Universal Robots URScript: samho_main_Fillet_2024_02_13.script

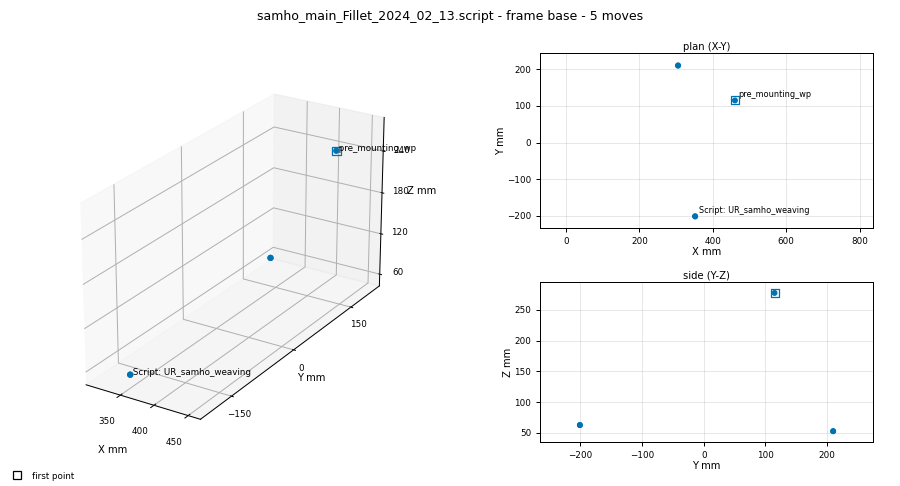
[picture p0: tool path of samho_main_Fillet_2024_02_13.script in frame base, 5 of 124 moves have a stored position in this frame; points joined in program order, loops and branches not executed]
def samho_main_Fillet_2024_02_13():
  step_count_5ae82350_5487_4ba1_a1cc_34982a72aa39 = 0.0
  thread Step_Counter_Thread_2c366939_5a87_4f2f_9225_c5964de88690():
    while (True):
      step_count_5ae82350_5487_4ba1_a1cc_34982a72aa39 = step_count_5ae82350_5487_4ba1_a1cc_34982a72aa39 + 1.0
      sync()
    end
  end
  run Step_Counter_Thread_2c366939_5a87_4f2f_9225_c5964de88690()
  modbus_add_signal("127.0.0.1", 255, 171, 2, "MODBUS_1", False)
  modbus_set_signal_update_frequency("MODBUS_1", 1)
  modbus_add_signal("127.0.0.1", 255, 153, 2, "MODBUS_2", False)
  modbus_set_signal_update_frequency("MODBUS_2", 10)
  modbus_add_signal("127.0.0.1", 255, 154, 2, "MODBUS_3", False)
  modbus_set_signal_update_frequency("MODBUS_3", 10)
  modbus_add_signal("127.0.0.1", 255, 240, 2, "MODBUS_4", False)
  modbus_set_signal_update_frequency("MODBUS_4", 10)
  set_safety_mode_transition_hardness(1)
  set_gravity([0.0, 0.0, 9.82])
  set_tool_voltage(24)
  set_tcp(p[-0.20862,-0.00524,0.38449,1.2551,0.019,-2.8747])
  set_payload(2.4, [-0.085, 0.00191, 0.125])
  set_standard_analog_input_domain(0, 1)
  set_standard_analog_input_domain(1, 1)
  set_tool_analog_input_domain(0, 1)
  set_tool_analog_input_domain(1, 1)
  set_analog_outputdomain(0, 1)
  set_analog_outputdomain(1, 1)
  set_input_actions_to_default()
  set_tool_digital_input_action(1, "freedrive")
  set_runstate_standard_digital_outputs([0])
  set_runstate_standard_digital_output_to_value(0, 1)
  set_runstate_standard_digital_output_to_value(7, 3)
  global A_Touch_trig_l=[False, True, False, True, True, True, False, True, False, False, False]
  global Auto_cur_cell=3
  global last_wv_line=p[0.52015, 0.38218, -0.0375, -1.74526, -0.73525, -1.7528]
  global Auto_trig=True
  global A_Touch_p=[p[0, 0, 0, 0, 0, 0], p[0.52015, 0.38218, -0.0375, -1.74526, -0.73525, -1.7528], p[0, 0, 0, 0, 0, 0], p[0.50413, -0.42159, 0.00426, 1.77234, -0.72849, 1.76591], p[0.52, -0.2132, 0.01111, 1.77234, -0.72849, 1.76591], p[0.51743, 0.37705, -0.04254, -1.78159, 1.77436, -0.70262], p[0, 0, 0, 0, 0, 0], p[0.52006, -0.30606, -0.04378, -1.76775, 1.766, -0.72811], p[0, 0, 0, 0, 0, 0], p[0, 0, 0, 0, 0, 0], p[0, 0, 0, 0, 0, 0], p[0, 0, 0, 0, 0, 0], p[0, 0, 0, 0, 0, 0], p[0, 0, 0, 0, 0, 0], p[0, 0, 0, 0, 0, 0], p[0, 0, 0, 0, 0, 0]]
  global last_wv_wp1=p[0.52015, 0.38218, -0.0375, -1.74526, -0.73525, -1.7528]
  global last_pose=p[0.52041, 0.38156, 0.01096, -2.11461, -0.89189, -1.42384]
  global A_Distance_list=[0, 0, 0, 0, 0, 0, 0, 0, 0, 0, 0, 0, 0, 0, 0, 0]
  global Auto_total_cell=5
  global A_Prepos_l=[p[0, 0, 0, 0, 0, 0], p[0.4924, 0.36901, -0.00027, -2.2158, -0.90076, -1.37843], p[0, 0, 0, 0, 0, 0], p[0.4524, -0.39099, 0.02973, 1.87806, -1.1242, 1.55521], p[0.4524, -0.16099, 0.02973, 1.87806, -1.1242, 1.55521], p[0.49166, 0.359, 0.00223, -2.36087, -1.03274, -1.30238], p[0, 0, 0, 0, 0, 0], p[0.45295, -0.28098, -0.02711, 2.2659, -1.09056, 1.27338], p[0, 0, 0, 0, 0, 0], p[0, 0, 0, 0, 0, 0], p[0, 0, 0, 0, 0, 0], p[0, 0, 0, 0, 0, 0], p[0, 0, 0, 0, 0, 0], p[0, 0, 0, 0, 0, 0], p[0, 0, 0, 0, 0, 0], p[0, 0, 0, 0, 0, 0]]
  global Reset_Trig=False
  global Auto_W_num=[4, 31, 32, 1, 3, 0, 0, 0, 0, 0, 0, 0, 0, 0, 0]
  global A_Speed_list=[0, 0, 0, 0, 0, 0, 0, 0, 0, 0, 0, 0, 0, 0, 0, 0]
  global last_z_bottom=-0.0502
  global last_tilt_deg=[0, -27, 0]
  global Base=p[0.0,0.0,0.0,0.0,0.0,0.0]
  global save_timer=0
  global timer_1=0
  def calculate_point_to_move_towards(feature, direction, position_distance):
    local posDir=[direction[0], direction[1], direction[2]]
    if (norm(posDir) < 1e-6):
      return get_target_waypoint()
    end
    local direction_vector_normalized=normalize(posDir)
    local displacement_pose=p[direction_vector_normalized[0] * position_distance,direction_vector_normalized[1] * position_distance,direction_vector_normalized[2] * position_distance,0,0,0]
    local wanted_displacement_in_base_frame=pose_sub(pose_trans(feature, displacement_pose), feature)
    return pose_add(get_target_waypoint(), wanted_displacement_in_base_frame)
  end
  global save_timer_is_counting=False
  global timer_1_is_counting=False
  thread Timer_Thread():
    while (True):
      if (save_timer_is_counting):
        save_timer = save_timer + get_steptime()
      end
      if (timer_1_is_counting):
        timer_1 = timer_1 + get_steptime()
      end
      sync()
    end
  end
  run Timer_Thread()
  def cell_info():
    $ 1514 "cell_info" "noBreak"
    $ 1515 "'cell_setting'"
    # 'cell_setting'
    $ 1516 "a7_f_distance≔get_center"
    global a7_f_distance=get_center
    $ 1517 "'dis + 125'"
    # 'dis + 125'
    $ 1518 "If simulation_mode"
    if (simulation_mode):
      $ 1519 "a6_f_height_l≔190"
      global a6_f_height_l=190
      $ 1520 "a6_f_height_r≔190"
      global a6_f_height_r=190
      $ 1521 "a6_f_width≔690"
      global a6_f_width=690
      $ 1522 "a6_callar_hor≔100"
      global a6_callar_hor=100
      $ 1523 "a6_callar_vert≔100"
      global a6_callar_vert=100
      $ 1524 "center_height≔50"
      global center_height=50
      $ 1525 "EXT_flag1≔integer_to_binary_list(2048)"
      global EXT_flag1= integer_to_binary_list (2048)
      $ 1526 "get_margin_z≔50"
      global get_margin_z=50
    else:
      $ 1527 "Else" "noBreak"
      $ 1528 "a6_f_height_l≔read_port_register(173)"
      global a6_f_height_l= read_port_register (173)
      $ 1529 "a6_f_height_r≔read_port_register(174)"
      global a6_f_height_r= read_port_register (174)
      $ 1530 "a6_f_width≔read_port_register(175)"
      global a6_f_width= read_port_register (175)
      $ 1531 "a6_callar_hor≔read_port_register(181)"
      global a6_callar_hor= read_port_register (181)
      $ 1532 "a6_callar_vert≔read_port_register(182)"
      global a6_callar_vert= read_port_register (182)
      $ 1533 "center_height≔read_port_register(237)"
      global center_height=read_port_register(237)
      $ 1534 "EXT_flag1≔integer_to_binary_list(read_port_register(179))"
      global EXT_flag1= integer_to_binary_list ( read_port_register (179))
      $ 1536 "get_margin_z≔read_port_register(238)"
      global get_margin_z=read_port_register(238)
      $ 1538 "If center_height>32765"
      if (center_height>32765):
        $ 1539 "center_height≔center_height-65535"
        global center_height=center_height-65535
      end
      $ 1540 "If get_margin_z>32765"
      if (get_margin_z>32765):
        $ 1541 "get_margin_z≔get_margin_z-65535"
        global get_margin_z=get_margin_z-65535
      end
    end
    $ 1542 "Initialization"
    $ 1543 "CELL_ROBOT_DIST≔a7_f_distance"
    global CELL_ROBOT_DIST=a7_f_distance
    $ 1544 "CELL_WIDTH≔a6_f_width"
    global CELL_WIDTH=a6_f_width
  end
  def robotand_cell_initalizat():
    $ 1545 "robotand_cell_initalizat" "noBreak"
    $ 1546 "If Auto_trig≟ True "
    if (Auto_trig ==   True  ):
      $ 1547 "Auto_trig≔ False "
      global Auto_trig=  False
      $ 1548 "init"
      $ 1549 "write_port_register(cell_3f_2f_151,0)"
      write_port_register(cell_3f_2f_151,0)
      $ 1550 "write_port_register(cell_info_152,0)"
      write_port_register(cell_info_152,0)
      $ 1551 "write_port_register(weld_req_153,0)"
      write_port_register(weld_req_153,0)
      $ 1552 "write_port_register(touch_cell_155,0)"
      write_port_register(touch_cell_155,0)
      $ 1553 "write_port_register(touch_num_156,0)"
      write_port_register(touch_num_156,0)
      $ 1554 "write_port_register(touch_done_157,0)"
      write_port_register(touch_done_157,0)
      $ 1555 "write_port_register(weld_done_137,0)"
      write_port_register(weld_done_137,0)
      $ 1556 "write_port_register(135,0)"
      write_port_register(135,0)
      $ 1557 "write_port_register(136,0)"
      write_port_register(136,0)
      $ 1558 "write_port_register(165,0)"
      write_port_register(165,0)
      $ 1559 "write_port_register(166,0)"
      write_port_register(166,0)
      $ 1560 "write_port_register(167,0)"
      write_port_register(167,0)
      $ 1561 "write_port_register(169,0)"
      write_port_register(169,0)
      $ 1562 "write_port_register(170,0)"
      write_port_register(170,0)
      $ 1563 "write_port_register(221,0)"
      write_port_register(221,0)
      $ 1564 "write_port_register(222,0)"
      write_port_register(222,0)
      $ 1565 "write_port_register(223,0)"
      write_port_register(223,0)
      $ 1566 "write_port_register(224,0)"
      write_port_register(224,0)
      $ 1567 "write_port_register(225,0)"
      write_port_register(225,0)
      $ 1568 "write_port_register(226,0)"
      write_port_register(226,0)
      $ 1569 "write_port_register(227,0)"
      write_port_register(227,0)
      $ 1570 "write_port_register(228,0)"
      write_port_register(228,0)
      $ 1571 "write_port_register(240,0)"
      write_port_register(240,0)
      $ 1572 "write_port_register(176,0)"
      write_port_register(176,0)
      $ 1573 "write_port_register(177,0)"
      write_port_register(177,0)
      $ 1574 "write_port_register(154,0)"
      write_port_register(154,0)
    end
    $ 1575 "sync()"
    sync()
  end
  def welding_parameter_init():
    $ 1576 "welding_parameter_init" "noBreak"
    $ 1577 "init"
    $ 1578 "If A_sel_v≟A_VL1 or A_sel_v≟A_VL2 or A_sel_v≟A_VR1 or A_sel_v≟A_VR2"
    if (A_sel_v == A_VL1  or  A_sel_v == A_VL2  or  A_sel_v == A_VR1  or  A_sel_v == A_VR2):
      $ 1579 "position_3f2f≔position_3F"
      global position_3f2f=position_3F
      $ 1580 "write_port_register(cell_3f_2f_151,A_sel_v)"
      write_port_register(cell_3f_2f_151,A_sel_v)
      $ 1581 "b8_wv_2f≔ False "
      global b8_wv_2f=  False
      $ 1582 "d_lean_degree≔0"
      global d_lean_degree=0
    else:
      $ 1583 "Else" "noBreak"
      $ 1584 "position_3f2f≔position_2F"
      global position_3f2f=position_2F
      $ 1585 "b8_wv_2f≔ True "
      global b8_wv_2f=  True
      $ 1586 "d_lean_degree≔30"
      global d_lean_degree=30
      $ 1587 "write_port_register(cell_3f_2f_151,A_HOR)"
      write_port_register(cell_3f_2f_151,A_HOR)
    end
    $ 1588 "If current_path≥2"
    if (current_path >= 2):
      $ 1589 "write_port_register(cell_info_152,current_path)"
      write_port_register(cell_info_152,current_path)
    else:
      $ 1590 "Else" "noBreak"
      $ 1591 "write_port_register(cell_info_152,1)"
      write_port_register(cell_info_152,1)
    end
    $ 1592 "write_port_register(return_done_240,0)"
    write_port_register(return_done_240,0)
    $ 1593 "Wait: 0.3"
    sleep(0.3)
    $ 1594 "write_port_register(weld_req_153,1)"
    write_port_register(weld_req_153,1)
    $ 1595 "Wait read_port_register(return_done_240)≟1"
    while (not( read_port_register (return_done_240) == 1)):
      sync()
    end
    $ 1596 "write_port_register(weld_req_153,0)"
    write_port_register(weld_req_153,0)
    $ 1597 "touch_m_check≔0"
    global touch_m_check=0
    $ 1598 "start_end_from_pendant"
    $ 1599 "d_start_current≔read_port_register(244)/10"
    global d_start_current= read_port_register (244)/10
    $ 1600 "d_start_voltage≔read_port_register(245)/10"
    global d_start_voltage= read_port_register (245)/10
    $ 1601 "d_start_time≔read_port_register(241)/10"
    global d_start_time= read_port_register (241)/10
    $ 1602 "d_end_current≔read_port_register(249)/10"
    global d_end_current= read_port_register (249)/10
    $ 1603 "d_end_voltage≔read_port_register(250)/10"
    global d_end_voltage= read_port_register (250)/10
    $ 1604 "d_end_time≔read_port_register(246)/10"
    global d_end_time= read_port_register (246)/10
    $ 1605 "d_end_current_2≔read_port_register(254)/10"
    global d_end_current_2= read_port_register (254)/10
    $ 1606 "d_end_voltage_2≔read_port_register(255)/10"
    global d_end_voltage_2= read_port_register (255)/10
    $ 1607 "d_end_time_2≔read_port_register(251)/10"
    global d_end_time_2= read_port_register (251)/10
    $ 1608 "a7_weld_crater≔[d_start_current,d_start_voltage,d_start_time,d_end_current,d_end_voltage,d_end_time,d_lean_degree]"
    global a7_weld_crater=[d_start_current,d_start_voltage,d_start_time,d_end_current,d_end_voltage,d_end_time,d_lean_degree]
    $ 1609 "a0_volt_ref≔read_port_register(231)/10"
    global a0_volt_ref= read_port_register (231)/10
    $ 1610 "a1_amp_ref≔read_port_register(232)/10"
    global a1_amp_ref= read_port_register (232)/10
    $ 1611 "a2_speed_cpm≔read_port_register(233)/10"
    global a2_speed_cpm= read_port_register (233)/10
    $ 1612 "a3_wv_amplitude≔read_port_register(234)/10"
    global a3_wv_amplitude= read_port_register (234)/10
    $ 1613 "a4_wv_frequency≔read_port_register(225)/10"
    global a4_wv_frequency= read_port_register (225)/10
    $ 1614 "b1_appro_param≔0"
    global b1_appro_param=0
    $ 1615 "b4_wv_delay2≔read_port_register(226)/10"
    global b4_wv_delay2= read_port_register (226)/10
    $ 1616 "b6_wv_delay4≔read_port_register(227)/10"
    global b6_wv_delay4= read_port_register (227)/10
    $ 1619 "b3_wv_delay1≔0"
    global b3_wv_delay1=0
    $ 1620 "b5_wv_delay3≔0"
    global b5_wv_delay3=0
    $ 1621 "b3_dealy_all≔[b3_wv_delay1,b4_wv_delay2,b5_wv_delay3,b6_wv_delay4]"
    global b3_dealy_all=[b3_wv_delay1,b4_wv_delay2,b5_wv_delay3,b6_wv_delay4]
    $ 1622 "get_width_182≔read_port_register(182)"
    global get_width_182= read_port_register (182)
    $ 1623 "b9_touch_sens≔20"
    global b9_touch_sens=20
    $ 1624 "task_angle≔register_read(228)/10"
    global task_angle=register_read(228)/10
    $ 1625 "Circle_Speed≔a2_speed_cpm"
    global Circle_Speed=a2_speed_cpm
    $ 1626 "CELL_BOTTOM≔a7_cell_bottom"
    global CELL_BOTTOM=a7_cell_bottom
    $ 1627 "a6_scallup_left≔read_port_register(176)"
    global a6_scallup_left= read_port_register (176)
    $ 1628 "a6_scallup_righ≔read_port_register(177)"
    global a6_scallup_righ= read_port_register (177)
    $ 1629 "a5_f_hole≔[a7_cell_bottom,a6_scallup_left,a6_scallup_righ]"
    global a5_f_hole=[a7_cell_bottom,a6_scallup_left,a6_scallup_righ]
    $ 1663 "폴더"
    $ 1664 "offset_2f_x≔7"
    global offset_2f_x=7
    $ 1665 "offset_3f_z≔-5"
    global offset_3f_z=-5
    $ 1666 "If A_sel_v≟A_VR1 or A_sel_v≟A_VR2"
    if (A_sel_v == A_VR1  or  A_sel_v == A_VR2):
      $ 1667 "'3F'"
      # '3F'
      $ 1668 "b2_left_par≔ False "
      global b2_left_par=  False
      $ 1669 "b8_wv_type≔1"
      global b8_wv_type=1
      $ 1670 "If A_sel_v≟A_VR2 and (b1_cell_info_R≟c or b1_cell_info_R≟d)"
      if (A_sel_v == A_VR2  and  (b1_cell_info_R == c  or  b1_cell_info_R == d)):
        $ 1671 "b7_tilt_degree≔[0,0,0]"
        global b7_tilt_degree=[0,0,0]
      else:
        $ 1672 "Else" "noBreak"
        $ 1673 "b7_tilt_degree≔[task_angle,-27,0]"
        global b7_tilt_degree=[task_angle,-27,0]
      end
      $ 1674 "c3_arc_enable≔1"
      global c3_arc_enable=1
    else:
      $ 1675 "ElseIf A_sel_v≟A_VL1 or A_sel_v≟A_VL2"
      if (A_sel_v == A_VL1  or  A_sel_v == A_VL2):
        $ 1676 "'3F'"
        # '3F'
        $ 1677 "b2_left_par≔ True "
        global b2_left_par=  True
        $ 1678 "b8_wv_type≔1"
        global b8_wv_type=1
        $ 1679 "If A_sel_v≟A_VL2 and (b1_cell_info_L≟c or b1_cell_info_L≟d)"
        if (A_sel_v == A_VL2  and  (b1_cell_info_L == c  or  b1_cell_info_L == d)):
          $ 1680 "b7_tilt_degree≔[0,0,0]"
          global b7_tilt_degree=[0,0,0]
        else:
          $ 1681 "Else" "noBreak"
          $ 1682 "b7_tilt_degree≔[task_angle,-27,0]"
          global b7_tilt_degree=[task_angle,-27,0]
        end
        $ 1683 "c3_arc_enable≔1"
        global c3_arc_enable=1
      else:
        $ 1684 "Else" "noBreak"
        $ 1685 "b2_left_par≔ True "
        global b2_left_par=  True
        $ 1686 "b8_wv_type≔2"
        global b8_wv_type=2
        $ 1687 "If A_sel_v≟A_HOR"
        if (A_sel_v == A_HOR):
          $ 1688 "b7_tilt_degree≔[30,-1*task_angle,0]"
          global b7_tilt_degree=[30,-1*task_angle,0]
        else:
          $ 1689 "Else" "noBreak"
          $ 1691 "b7_tilt_degree≔[30,-1*task_angle,0]"
          global b7_tilt_degree=[30,-1*task_angle,0]
        end
        $ 1693 "c3_arc_enable≔0"
        global c3_arc_enable=0
      end
    end
    $ 1694 "If A_sel_v≟A_VL2 or A_sel_v≟A_VR2"
    if (A_sel_v == A_VL2  or  A_sel_v == A_VR2):
      $ 1695 "If b1_cell_info_L≟E or b1_cell_info_L≟e or b1_cell_info_R≟E or b1_cell_info_R≟e"
      if (b1_cell_info_L == E  or  b1_cell_info_L == e  or  b1_cell_info_R == E  or  b1_cell_info_R == e):
        $ 1696 "a8_wv_distance≔read_port_register(182)-a5_f_hole[1]-offset_3f_begin"
        global a8_wv_distance= read_port_register (182)-a5_f_hole[1]-offset_3f_begin
      else:
        $ 1697 "Else" "noBreak"
        $ 1698 "a8_wv_distance≔read_port_register(182)-offset_3f_begin"
        global a8_wv_distance= read_port_register (182)-offset_3f_begin
      end
    else:
      $ 1703 "Else" "noBreak"
      $ 1704 "If b2_left_par"
      if (b2_left_par):
        $ 1705 "Comment"
        # Comment
        $ 1706 "a8_wv_distance≔a6_f_height_l-a5_f_hole[1]-offset_3f_begin"
        global a8_wv_distance=a6_f_height_l-a5_f_hole[1]-offset_3f_begin
        $ 1707 "Comment"
        # Comment
      else:
        $ 1708 "Else" "noBreak"
        $ 1709 "a8_wv_distance≔a6_f_height_r-a5_f_hole[1]-offset_3f_begin"
        global a8_wv_distance=a6_f_height_r-a5_f_hole[1]-offset_3f_begin
      end
    end
    $ 1710 "Ext fun & Squash"
    $ 1711 "If (A_sel_v≟A_VL1 or A_sel_v≟A_VL2) and (b1_cell_info_L≟B or b1_cell_info_L≟D)"
    if ((A_sel_v == A_VL1  or  A_sel_v == A_VL2)  and  (b1_cell_info_L == B  or  b1_cell_info_L == D)):
      $ 1712 "Scallup_check≔ True "
      global Scallup_check=  True
    else:
      $ 1713 "ElseIf (A_sel_v≟A_VR1 or A_sel_v≟A_VR2) and (b1_cell_info_R≟B or b1_cell_info_R≟D)"
      if ((A_sel_v == A_VR1  or  A_sel_v == A_VR2)  and  (b1_cell_info_R == B  or  b1_cell_info_R == D)):
        $ 1714 "Scallup_check≔ True "
        global Scallup_check=  True
      else:
        $ 1715 "Else" "noBreak"
        $ 1716 "Scallup_check≔ False "
        global Scallup_check=  False
      end
    end
    $ 1717 "'squash'"
    # 'squash'
    $ 1718 "If (EXT_flag1[7]≟ True ) and (A_sel_v≠A_HOR) and (A_sel_v≠A_VL2) and (A_sel_v≠A_VR2) and (Scallup_check≟ False ) and (A_sel_v≟A_VL1 and b1_cell_info_L≠E and b1_cell_info_L≠e) and (A_sel_v≟A_VR1 and b1_cell_info_R≠E and b1_cell_info_R≠e)"
    if ((EXT_flag1[7] ==   True  )  and  (A_sel_v != A_HOR)  and  (A_sel_v != A_VL2)  and  (A_sel_v != A_VR2)  and  (Scallup_check ==   False  )  and  (A_sel_v == A_VL1  and  b1_cell_info_L != E  and  b1_cell_info_L != e)  and  (A_sel_v == A_VR1  and  b1_cell_info_R != E  and  b1_cell_info_R != e)):
      $ 1719 "squash"
      $ 1720 "squash_enable≔1"
      global squash_enable=1
      $ 1721 "squash_voltage≔24.5"
      global squash_voltage=24.5
      $ 1722 "squash_current≔190"
      global squash_current=190
      $ 1723 "squash_amp≔7"
      global squash_amp=7
      $ 1724 "squash_speed≔10"
      global squash_speed=10
      $ 1725 "squash_cycle≔8"
      global squash_cycle=8
    else:
      $ 1726 "Else" "noBreak"
      $ 1727 "squash"
      $ 1728 "squash_enable≔0"
      global squash_enable=0
      $ 1729 "squash_voltage≔0"
      global squash_voltage=0
      $ 1730 "squash_current≔0"
      global squash_current=0
      $ 1731 "squash_amp≔0"
      global squash_amp=0
      $ 1732 "squash_speed≔0"
      global squash_speed=0
      $ 1733 "squash_cycle≔0"
      global squash_cycle=0
    end
    $ 1734 "'sladge'"
    # 'sladge'
    $ 1735 "If EXT_flag1[8]≟ True  and EXT_flag1[9]≟ False "
    if (EXT_flag1[8] ==   True    and  EXT_flag1[9] ==   False  ):
      $ 1736 "sludge≔1"
      global sludge=1
    else:
      $ 1737 "ElseIf EXT_flag1[8]≟ False  and EXT_flag1[9]≟ True "
      if (EXT_flag1[8] ==   False    and  EXT_flag1[9] ==   True  ):
        $ 1738 "sludge≔2"
        global sludge=2
      else:
        $ 1739 "Else" "noBreak"
        $ 1740 "sludge≔0"
        global sludge=0
      end
    end
    $ 1741 "waste_cycle≔2"
    global waste_cycle=2
    $ 1742 "c0_offset_x≔read_port_register(229)/10"
    global c0_offset_x= read_port_register (229)/10
    $ 1743 "c0_offset_z≔read_port_register(230)/10"
    global c0_offset_z= read_port_register (230)/10
    $ 1744 "squash_l≔[a0_volt_ref,a1_amp_ref,squash_enable,squash_voltage,squash_current,squash_amp,squash_speed,squash_cycle,waste_cycle,c0_offset_x,c0_offset_z]"
    global squash_l=[a0_volt_ref,a1_amp_ref,squash_enable,squash_voltage,squash_current,squash_amp,squash_speed,squash_cycle,waste_cycle,c0_offset_x,c0_offset_z]
    $ 1745 "WV_gap"
    $ 1746 "c5_wv_gap_y≔read_port_register(236)/10"
    global c5_wv_gap_y= read_port_register (236)/10
    $ 1747 "c6_wv_gap_cpm≔read_port_register(235)/10"
    global c6_wv_gap_cpm= read_port_register (235)/10
    $ 1748 "c9_wv_gap_freq≔a4_wv_frequency"
    global c9_wv_gap_freq=a4_wv_frequency
    $ 1749 "If c6_wv_gap_cpm≟a2_speed_cpm and a3_wv_amplitude≟c5_wv_gap_y"
    if (c6_wv_gap_cpm == a2_speed_cpm  and  a3_wv_amplitude == c5_wv_gap_y):
      $ 1750 "c4_gap_enable≔0"
      global c4_gap_enable=0
    else:
      $ 1751 "Else" "noBreak"
      $ 1752 "c4_gap_enable≔1"
      global c4_gap_enable=1
    end
    $ 1753 "c7_wv_gap≔[c4_gap_enable,c5_wv_gap_y,c6_wv_gap_cpm,c9_wv_gap_freq]"
    global c7_wv_gap=[c4_gap_enable,c5_wv_gap_y,c6_wv_gap_cpm,c9_wv_gap_freq]
    $ 1754 "arc_sen"
    $ 1755 "c3_X_p_gain≔read_port_register(186)/10"
    global c3_X_p_gain= read_port_register (186)/10
    $ 1756 "c3_X_i_gain≔read_port_register(187)/10"
    global c3_X_i_gain= read_port_register (187)/10
    $ 1757 "c3_Z_p_gain≔read_port_register(184)/10"
    global c3_Z_p_gain= read_port_register (184)/10
    $ 1758 "c3_Z_i_gain≔read_port_register(185)/10"
    global c3_Z_i_gain= read_port_register (185)/10
    $ 1759 "c3_wv_arc_fix≔0"
    global c3_wv_arc_fix=0
    $ 1760 "c3_wv_arc≔[c3_arc_enable,c3_X_p_gain,c3_X_i_gain,c3_Z_p_gain,c3_Z_i_gain,c3_wv_arc_fix]"
    global c3_wv_arc=[c3_arc_enable,c3_X_p_gain,c3_X_i_gain,c3_Z_p_gain,c3_Z_i_gain,c3_wv_arc_fix]
    $ 1761 "volt and current"
    $ 1762 "set_current_voltage(a1_amp_ref,a0_volt_ref)"
    set_current_voltage(a1_amp_ref,a0_volt_ref)
    $ 1763 "write_port_register(154,1)"
    write_port_register(154,1)
    $ 1764 "Wait read_port_register(return_done_240)≟0"
    while (not( read_port_register (return_done_240) == 0)):
      sync()
    end
    $ 1765 "write_port_register(154,0)"
    write_port_register(154,0)
  end
  def welding_parameter_sim():
    $ 1766 "welding_parameter_sim" "noBreak"
    $ 1767 "init"
    $ 1768 "If A_sel_v≟A_VL1 or A_sel_v≟A_VL2 or A_sel_v≟A_VR1 or A_sel_v≟A_VR2"
    if (A_sel_v == A_VL1  or  A_sel_v == A_VL2  or  A_sel_v == A_VR1  or  A_sel_v == A_VR2):
      $ 1769 "position_3f2f≔position_3F"
      global position_3f2f=position_3F
      $ 1770 "write_port_register(cell_3f_2f_151,A_sel_v)"
      write_port_register(cell_3f_2f_151,A_sel_v)
      $ 1771 "b8_wv_2f≔ False "
      global b8_wv_2f=  False
      $ 1772 "d_lean_degree≔0"
      global d_lean_degree=0
    else:
      $ 1773 "Else" "noBreak"
      $ 1774 "position_3f2f≔position_2F"
      global position_3f2f=position_2F
      $ 1775 "b8_wv_2f≔ True "
      global b8_wv_2f=  True
      $ 1776 "d_lean_degree≔30"
      global d_lean_degree=30
      $ 1777 "write_port_register(cell_3f_2f_151,A_HOR)"
      write_port_register(cell_3f_2f_151,A_HOR)
    end
    $ 1778 "If current_path≥2"
    if (current_path >= 2):
      $ 1779 "write_port_register(cell_info_152,current_path)"
      write_port_register(cell_info_152,current_path)
    else:
      $ 1780 "Else" "noBreak"
      $ 1781 "write_port_register(cell_info_152,1)"
      write_port_register(cell_info_152,1)
    end
    $ 1782 "write_port_register(return_done_240,0)"
    write_port_register(return_done_240,0)
    $ 1783 "Wait: 0.3"
    sleep(0.3)
    $ 1784 "write_port_register(weld_req_153,1)"
    write_port_register(weld_req_153,1)
    $ 1786 "write_port_register(weld_req_153,0)"
    write_port_register(weld_req_153,0)
    $ 1787 "touch_m_check≔0"
    global touch_m_check=0
    $ 1788 "start_end_from_pendant"
    $ 1789 "d_start_current≔read_port_register(244)/10"
    global d_start_current= read_port_register (244)/10
    $ 1790 "d_start_voltage≔read_port_register(245)/10"
    global d_start_voltage= read_port_register (245)/10
    $ 1791 "d_start_time≔read_port_register(241)/10"
    global d_start_time= read_port_register (241)/10
    $ 1792 "d_end_current≔read_port_register(249)/10"
    global d_end_current= read_port_register (249)/10
    $ 1793 "d_end_voltage≔read_port_register(250)/10"
    global d_end_voltage= read_port_register (250)/10
    $ 1794 "d_end_time≔read_port_register(246)/10"
    global d_end_time= read_port_register (246)/10
    $ 1795 "d_end_current_2≔read_port_register(254)/10"
    global d_end_current_2= read_port_register (254)/10
    $ 1796 "d_end_voltage_2≔read_port_register(255)/10"
    global d_end_voltage_2= read_port_register (255)/10
    $ 1797 "d_end_time_2≔read_port_register(251)/10"
    global d_end_time_2= read_port_register (251)/10
    $ 1798 "a7_weld_crater≔[d_start_current,d_start_voltage,d_start_time,d_end_current,d_end_voltage,d_end_time,d_lean_degree]"
    global a7_weld_crater=[d_start_current,d_start_voltage,d_start_time,d_end_current,d_end_voltage,d_end_time,d_lean_degree]
    $ 1799 "a0_volt_ref≔read_port_register(231)/10"
    global a0_volt_ref= read_port_register (231)/10
    $ 1800 "a1_amp_ref≔read_port_register(232)/10"
    global a1_amp_ref= read_port_register (232)/10
    $ 1801 "b1_appro_param≔0"
    global b1_appro_param=0
    $ 1802 "Folder"
    $ 1803 "a2_speed_cpm≔17"
    global a2_speed_cpm=17
    $ 1804 "a3_wv_amplitude≔5"
    global a3_wv_amplitude=5
    $ 1805 "a4_wv_frequency≔1.4"
    global a4_wv_frequency=1.4
    $ 1806 "b4_wv_delay2≔0.3"
    global b4_wv_delay2=0.3
    $ 1807 "b6_wv_delay4≔0.3"
    global b6_wv_delay4=0.3
    $ 1808 "b9_touch_sens≔10"
    global b9_touch_sens=10
    $ 1809 "task_angle≔0"
    global task_angle=0
    $ 1810 "a6_scallup_left≔0"
    global a6_scallup_left=0
    $ 1811 "a6_scallup_righ≔0"
    global a6_scallup_righ=0
    $ 1812 "b3_wv_delay1≔0"
    global b3_wv_delay1=0
    $ 1813 "b5_wv_delay3≔0"
    global b5_wv_delay3=0
    $ 1814 "b3_dealy_all≔[b3_wv_delay1,b4_wv_delay2,b5_wv_delay3,b6_wv_delay4]"
    global b3_dealy_all=[b3_wv_delay1,b4_wv_delay2,b5_wv_delay3,b6_wv_delay4]
    $ 1815 "get_width_182≔a6_callar_vert"
    global get_width_182=a6_callar_vert
    $ 1816 "task_angle≔register_read(228)/10"
    global task_angle=register_read(228)/10
    $ 1817 "Circle_Speed≔a2_speed_cpm"
    global Circle_Speed=a2_speed_cpm
    $ 1818 "CELL_BOTTOM≔a7_cell_bottom"
    global CELL_BOTTOM=a7_cell_bottom
    $ 1819 "a5_f_hole≔[a7_cell_bottom,a6_scallup_left,a6_scallup_righ]"
    global a5_f_hole=[a7_cell_bottom,a6_scallup_left,a6_scallup_righ]
    $ 1820 "폴더"
    $ 1821 "offset_2f_x≔7"
    global offset_2f_x=7
    $ 1822 "offset_3f_z≔-5"
    global offset_3f_z=-5
    $ 1823 "If A_sel_v≟A_VR1 or A_sel_v≟A_VR2"
    if (A_sel_v == A_VR1  or  A_sel_v == A_VR2):
      $ 1824 "'3F'"
      # '3F'
      $ 1825 "b2_left_par≔ False "
      global b2_left_par=  False
      $ 1826 "b8_wv_type≔1"
      global b8_wv_type=1
      $ 1827 "b7_tilt_degree≔[task_angle,-27,0]"
      global b7_tilt_degree=[task_angle,-27,0]
      $ 1828 "c3_arc_enable≔1"
      global c3_arc_enable=1
    else:
      $ 1829 "ElseIf A_sel_v≟A_VL1 or A_sel_v≟A_VL2"
      if (A_sel_v == A_VL1  or  A_sel_v == A_VL2):
        $ 1830 "'3F'"
        # '3F'
        $ 1831 "b2_left_par≔ True "
        global b2_left_par=  True
        $ 1832 "b8_wv_type≔1"
        global b8_wv_type=1
        $ 1833 "b7_tilt_degree≔[task_angle,-27,0]"
        global b7_tilt_degree=[task_angle,-27,0]
        $ 1834 "c3_arc_enable≔1"
        global c3_arc_enable=1
      else:
        $ 1835 "Else" "noBreak"
        $ 1836 "b2_left_par≔ True "
        global b2_left_par=  True
        $ 1837 "b8_wv_type≔2"
        global b8_wv_type=2
        $ 1838 "b7_tilt_degree≔[30,-1*task_angle,0]"
        global b7_tilt_degree=[30,-1*task_angle,0]
        $ 1840 "c3_arc_enable≔0"
        global c3_arc_enable=0
      end
    end
    $ 1841 "If A_sel_v≟A_VL2 or A_sel_v≟A_VR2"
    if (A_sel_v == A_VL2  or  A_sel_v == A_VR2):
      $ 1842 "a8_wv_distance≔read_port_register(182)"
      global a8_wv_distance= read_port_register (182)
    else:
      $ 1847 "Else" "noBreak"
      $ 1848 "If b2_left_par"
      if (b2_left_par):
        $ 1849 "Comment"
        # Comment
        $ 1850 "a8_wv_distance≔a6_f_height_l-a5_f_hole[1]"
        global a8_wv_distance=a6_f_height_l-a5_f_hole[1]
        $ 1851 "Comment"
        # Comment
      else:
        $ 1852 "Else" "noBreak"
        $ 1853 "a8_wv_distance≔a6_f_height_r-a5_f_hole[1]"
        global a8_wv_distance=a6_f_height_r-a5_f_hole[1]
      end
    end
    $ 1854 "Ext fun & Squash"
    $ 1855 "If (A_sel_v≟A_VL1 or A_sel_v≟A_VL2) and (b1_cell_info_L≟B or b1_cell_info_L≟D)"
    if ((A_sel_v == A_VL1  or  A_sel_v == A_VL2)  and  (b1_cell_info_L == B  or  b1_cell_info_L == D)):
      $ 1856 "Scallup_check≔ True "
      global Scallup_check=  True
    else:
      $ 1857 "ElseIf (A_sel_v≟A_VR1 or A_sel_v≟A_VR2) and (b1_cell_info_R≟B or b1_cell_info_R≟D)"
      if ((A_sel_v == A_VR1  or  A_sel_v == A_VR2)  and  (b1_cell_info_R == B  or  b1_cell_info_R == D)):
        $ 1858 "Scallup_check≔ True "
        global Scallup_check=  True
      else:
        $ 1859 "Else" "noBreak"
        $ 1860 "Scallup_check≔ False "
        global Scallup_check=  False
      end
    end
    $ 1861 "If (EXT_flag1[7]≟ True ) and (A_sel_v≠A_HOR) and (A_sel_v≠A_VL2) and (A_sel_v≠A_VR2) and (Scallup_check≟ False )"
    if ((EXT_flag1[7] ==   True  )  and  (A_sel_v != A_HOR)  and  (A_sel_v != A_VL2)  and  (A_sel_v != A_VR2)  and  (Scallup_check ==   False  )):
      $ 1862 "squash"
      $ 1863 "squash_enable≔1"
      global squash_enable=1
      $ 1864 "squash_voltage≔24.5"
      global squash_voltage=24.5
      $ 1865 "squash_current≔190"
      global squash_current=190
      $ 1866 "squash_amp≔7"
      global squash_amp=7
      $ 1867 "squash_speed≔10"
      global squash_speed=10
      $ 1868 "squash_cycle≔8"
      global squash_cycle=8
    else:
      $ 1869 "Else" "noBreak"
      $ 1870 "squash"
      $ 1871 "squash_enable≔0"
      global squash_enable=0
      $ 1872 "squash_voltage≔0"
      global squash_voltage=0
      $ 1873 "squash_current≔0"
      global squash_current=0
      $ 1874 "squash_amp≔0"
      global squash_amp=0
      $ 1875 "squash_speed≔0"
      global squash_speed=0
      $ 1876 "squash_cycle≔0"
      global squash_cycle=0
    end
    $ 1877 "waste_cycle≔2"
    global waste_cycle=2
    $ 1878 "c0_offset_x≔read_port_register(229)/10"
    global c0_offset_x= read_port_register (229)/10
    $ 1879 "c0_offset_z≔read_port_register(230)/10"
    global c0_offset_z= read_port_register (230)/10
    $ 1880 "squash_l≔[a0_volt_ref,a1_amp_ref,squash_enable,squash_voltage,squash_current,squash_amp,squash_speed,squash_cycle,waste_cycle,c0_offset_x,c0_offset_z]"
    global squash_l=[a0_volt_ref,a1_amp_ref,squash_enable,squash_voltage,squash_current,squash_amp,squash_speed,squash_cycle,waste_cycle,c0_offset_x,c0_offset_z]
    $ 1881 "WV_gap"
    $ 1882 "c5_wv_gap_y≔a3_wv_amplitude"
    global c5_wv_gap_y=a3_wv_amplitude
    $ 1883 "c6_wv_gap_cpm≔a2_speed_cpm"
    global c6_wv_gap_cpm=a2_speed_cpm
    $ 1884 "c9_wv_gap_freq≔a4_wv_frequency"
    global c9_wv_gap_freq=a4_wv_frequency
    $ 1885 "If c6_wv_gap_cpm≟a2_speed_cpm and a3_wv_amplitude≟c5_wv_gap_y"
    if (c6_wv_gap_cpm == a2_speed_cpm  and  a3_wv_amplitude == c5_wv_gap_y):
      $ 1886 "c4_gap_enable≔0"
      global c4_gap_enable=0
    else:
      $ 1887 "Else" "noBreak"
      $ 1888 "c4_gap_enable≔1"
      global c4_gap_enable=1
    end
    $ 1889 "c4_gap_enable≔0"
    global c4_gap_enable=0
    $ 1890 "c7_wv_gap≔[c4_gap_enable,c5_wv_gap_y,c6_wv_gap_cpm,c9_wv_gap_freq]"
    global c7_wv_gap=[c4_gap_enable,c5_wv_gap_y,c6_wv_gap_cpm,c9_wv_gap_freq]
    $ 1891 "arc_sen"
    $ 1892 "c3_X_p_gain≔read_port_register(186)/10"
    global c3_X_p_gain= read_port_register (186)/10
    $ 1893 "c3_X_i_gain≔read_port_register(187)/10"
    global c3_X_i_gain= read_port_register (187)/10
    $ 1894 "c3_Z_p_gain≔read_port_register(184)/10"
    global c3_Z_p_gain= read_port_register (184)/10
    $ 1895 "c3_Z_i_gain≔read_port_register(185)/10"
    global c3_Z_i_gain= read_port_register (185)/10
    $ 1896 "c3_wv_arc_fix≔0"
    global c3_wv_arc_fix=0
    $ 1897 "c3_wv_arc≔[c3_arc_enable,c3_X_p_gain,c3_X_i_gain,c3_Z_p_gain,c3_Z_i_gain,c3_wv_arc_fix]"
    global c3_wv_arc=[c3_arc_enable,c3_X_p_gain,c3_X_i_gain,c3_Z_p_gain,c3_Z_i_gain,c3_wv_arc_fix]
    $ 1898 "volt and current"
    $ 1899 "set_current_voltage(a1_amp_ref,a0_volt_ref)"
    set_current_voltage(a1_amp_ref,a0_volt_ref)
    $ 1900 "write_port_register(154,1)"
    write_port_register(154,1)
    $ 1902 "write_port_register(154,0)"
    write_port_register(154,0)
  end
  def Move_done():
    $ 1903 "Move_done" "noBreak"
    $ 1904 "write_port_register(robot_move_163,0)"
    write_port_register(robot_move_163,0)
    $ 1905 "write_port_register(robot_pose_164,0)"
    write_port_register(robot_pose_164,0)
    $ 1906 "write_port_register(robot_ready_141,1)"
    write_port_register(robot_ready_141,1)
  end
  def MoveFun():
    $ 1907 "MoveFun" "noBreak"
    $ 1908 "b_touch_pos≔A_Prepos_l[A_sel_v]"
    global b_touch_pos=A_Prepos_l[A_sel_v]
    $ 1909 "MoveL"
    $ 1910 "b_touch_pos" "breakAfter"
    movel(pose_trans(Base, b_touch_pos), a=0.35, v=0.35)
  end
  def MoveFun_cd():
    $ 1911 "MoveFun_cd" "noBreak"
    $ 1912 "b_touch_pos≔A_Prepos_l[A_sel_v]"
    global b_touch_pos=A_Prepos_l[A_sel_v]
    $ 1913 "If A_sel_v≟A_VR2 and (b1_cell_info_R≟c or b1_cell_info_R≟d)"
    if (A_sel_v == A_VR2  and  (b1_cell_info_R == c  or  b1_cell_info_R == d)):
      $ 1914 "tilt_deg≔27"
      global tilt_deg=27
      $ 1915 "tilt_deg_ry≔19"
      global tilt_deg_ry=19
      $ 1916 "tilt_deg_rz≔0"
      global tilt_deg_rz=0
    else:
      $ 1917 "Else" "noBreak"
      $ 1918 "tilt_deg≔10"
      global tilt_deg=10
      $ 1919 "tilt_deg_ry≔5"
      global tilt_deg_ry=5
      $ 1920 "tilt_deg_rz≔0"
      global tilt_deg_rz=0
    end
    $ 1921 "If b2_left_par"
    if (b2_left_par):
      $ 1922 "b_touch_pos≔pose_add(b_touch_pos, p[0,18/1000,0,0,0,0])"
      global b_touch_pos= pose_add (b_touch_pos, p[0,18/1000,0,0,0,0])
      $ 1923 "b_touch_pos≔pose_trans(b_touch_pos, p[0,0,0,d2r(-tilt_deg),d2r(-tilt_deg_ry),d2r(tilt_deg_rz)])"
      global b_touch_pos= pose_trans (b_touch_pos, p[0,0,0,d2r(-tilt_deg),d2r(-tilt_deg_ry),d2r(tilt_deg_rz)])
    else:
      $ 1924 "Else" "noBreak"
      $ 1925 "b_touch_pos≔pose_add(b_touch_pos, p[0,-18/1000,0,0,0,0])"
      global b_touch_pos= pose_add (b_touch_pos, p[0,-18/1000,0,0,0,0])
      $ 1926 "b_touch_pos≔pose_trans(b_touch_pos, p[0,0,0,d2r(tilt_deg),d2r(-tilt_deg_ry),d2r(-tilt_deg_rz)])"
      global b_touch_pos= pose_trans (b_touch_pos, p[0,0,0,d2r(tilt_deg),d2r(-tilt_deg_ry),d2r(-tilt_deg_rz)])
    end
    $ 1927 "MoveL"
    $ 1928 "b_touch_pos" "breakAfter"
    movel(pose_trans(Base, b_touch_pos), a=0.35, v=0.35)
  end
  def MoveandTouchFun_2f():
    $ 1929 "MoveandTouchFun_2f" "noBreak"
    $ 1930 "b_touch_pos≔A_Prepos_l[A_sel_v]"
    global b_touch_pos=A_Prepos_l[A_sel_v]
    $ 1931 "tilt_deg≔3"
    global tilt_deg=3
    $ 1932 "tilt_deg_ry≔3"
    global tilt_deg_ry=3
    $ 1933 "tilt_deg_rz≔0"
    global tilt_deg_rz=0
    $ 1934 "If  False "
    if (  False  ):
      $ 1935 "Wait: 0.01"
      sleep(0.01)
    else:
      $ 1936 "ElseIf A_sel_v≟A_HOR and b1_cell_info_L≟E"
      if (A_sel_v == A_HOR  and  b1_cell_info_L == E):
        $ 1937 "tilt_deg≔6"
        global tilt_deg=6
        $ 1938 "tilt_deg_ry≔-5"
        global tilt_deg_ry=-5
        $ 1939 "tilt_deg_rz≔0"
        global tilt_deg_rz=0
        $ 1940 "b_touch_pos≔pose_trans(b_touch_pos, p[0,0/1000,0,d2r(tilt_deg),d2r(-tilt_deg_ry),d2r(tilt_deg_rz)])"
        global b_touch_pos= pose_trans (b_touch_pos, p[0,0/1000,0,d2r(tilt_deg),d2r(-tilt_deg_ry),d2r(tilt_deg_rz)])
      else:
        $ 1941 "ElseIf A_sel_v≟A_HOR_R and b1_cell_info_R≟E"
        if (A_sel_v == A_HOR_R  and  b1_cell_info_R == E):
          $ 1942 "tilt_deg≔6"
          global tilt_deg=6
          $ 1943 "tilt_deg_ry≔-5"
          global tilt_deg_ry=-5
          $ 1944 "tilt_deg_rz≔0"
          global tilt_deg_rz=0
          $ 1945 "b_touch_pos≔pose_trans(b_touch_pos, p[0,0/1000,0,d2r(tilt_deg),d2r(-tilt_deg_ry),d2r(-tilt_deg_rz)])"
          global b_touch_pos= pose_trans (b_touch_pos, p[0,0/1000,0,d2r(tilt_deg),d2r(-tilt_deg_ry),d2r(-tilt_deg_rz)])
        else:
          $ 1946 "ElseIf b2_left_par"
          if (b2_left_par):
            $ 1947 "b_touch_pos≔pose_trans(b_touch_pos, p[0,0/1000,0,d2r(tilt_deg),d2r(-tilt_deg_ry),d2r(tilt_deg_rz)])"
            global b_touch_pos= pose_trans (b_touch_pos, p[0,0/1000,0,d2r(tilt_deg),d2r(-tilt_deg_ry),d2r(tilt_deg_rz)])
          else:
            $ 1948 "Else" "noBreak"
            $ 1949 "b_touch_pos≔pose_trans(b_touch_pos, p[0,0/1000,0,d2r(tilt_deg),d2r(-tilt_deg_ry),d2r(-tilt_deg_rz)])"
            global b_touch_pos= pose_trans (b_touch_pos, p[0,0/1000,0,d2r(tilt_deg),d2r(-tilt_deg_ry),d2r(-tilt_deg_rz)])
          end
        end
      end
    end
    $ 1950 "MoveL"
    $ 1951 "b_touch_pos" "breakAfter"
    movel(pose_trans(Base, b_touch_pos), a=0.35, v=0.35)
    $ 1952 "Touch_2f"
    $ 1953 "If  False "
    if (  False  ):
      $ 1954 "Wait: 0.01"
      sleep(0.01)
    else:
      $ 1955 "ElseIf A_sel_v≟A_HOR and b1_cell_info_L≟E"
      if (A_sel_v == A_HOR  and  b1_cell_info_L == E):
        $ 1956 "tilt_deg≔3"
        global tilt_deg=3
        $ 1957 "tilt_deg_ry≔3"
        global tilt_deg_ry=3
        $ 1958 "tilt_deg_rz≔0"
        global tilt_deg_rz=0
        $ 1959 "b_touch_pos2≔pose_trans(b_touch_pos, p[0,0/1000,0,d2r(tilt_deg),d2r(-tilt_deg_ry),d2r(tilt_deg_rz)])"
        global b_touch_pos2= pose_trans (b_touch_pos, p[0,0/1000,0,d2r(tilt_deg),d2r(-tilt_deg_ry),d2r(tilt_deg_rz)])
        $ 1960 "touch_result≔touch_fun_2f(b_touch_pos,b_touch_pos2,b2_left_par,b9_touch_sens)"
        global touch_result=touch_fun_2f(b_touch_pos,b_touch_pos2,b2_left_par,b9_touch_sens)
      else:
        $ 1961 "ElseIf A_sel_v≟A_HOR_R and b1_cell_info_R≟E"
        if (A_sel_v == A_HOR_R  and  b1_cell_info_R == E):
          $ 1962 "tilt_deg≔3"
          global tilt_deg=3
          $ 1963 "tilt_deg_ry≔3"
          global tilt_deg_ry=3
          $ 1964 "tilt_deg_rz≔0"
          global tilt_deg_rz=0
          $ 1965 "b_touch_pos2≔pose_trans(b_touch_pos, p[0,0/1000,0,d2r(tilt_deg),d2r(-tilt_deg_ry),d2r(-tilt_deg_rz)])"
          global b_touch_pos2= pose_trans (b_touch_pos, p[0,0/1000,0,d2r(tilt_deg),d2r(-tilt_deg_ry),d2r(-tilt_deg_rz)])
          $ 1966 "touch_result≔touch_fun_2f(b_touch_pos,b_touch_pos2,b2_left_par,b9_touch_sens)"
          global touch_result=touch_fun_2f(b_touch_pos,b_touch_pos2,b2_left_par,b9_touch_sens)
        else:
          $ 1967 "Else" "noBreak"
          $ 1968 "touch_result≔touch_fun_2f(b_touch_pos,b_touch_pos,b2_left_par,b9_touch_sens)"
          global touch_result=touch_fun_2f(b_touch_pos,b_touch_pos,b2_left_par,b9_touch_sens)
        end
      end
    end
    $ 1970 "If b2_left_par"
    if (b2_left_par):
      $ 1971 "touch_result≔pose_trans(touch_result,p[-(Touch_dis)/1000,0,0,0,0,0])"
      global touch_result= pose_trans (touch_result,p[-(Touch_dis)/1000,0,0,0,0,0])
    else:
      $ 1972 "Else" "noBreak"
      $ 1973 "touch_result≔pose_trans(touch_result,p[(Touch_dis)/1000,0,0,0,0,0])"
      global touch_result= pose_trans (touch_result,p[(Touch_dis)/1000,0,0,0,0,0])
    end
    $ 1974 "A_Touch_p[A_sel_v]=touch_result"
    A_Touch_p[A_sel_v]=touch_result
    $ 1975 "If EXT_flag1[3]≟ True "
    if (EXT_flag1[3] ==   True  ):
      $ 1976 "MoveL"
      $ 1977 "manual_tp≔tilt_2f_fun(touch_result,basic_tilt_2f,wv_direction)"
      global manual_tp=tilt_2f_fun(touch_result,basic_tilt_2f,wv_direction)
      $ 1978 "manual_tp≔pose_trans(manual_tp, p[0,0,-10/1000,0,0,0])"
      global manual_tp= pose_trans (manual_tp, p[0,0,-10/1000,0,0,0])
      $ 1979 "manual_tp" "breakAfter"
      movel(pose_trans(Base, manual_tp), a=0.3, v=0.15)
      $ 1980 "Wait: 1.5"
      sleep(1.5)
    end
  end
  def MoveandTouchFun_3f():
    $ 1981 "MoveandTouchFun_3f" "noBreak"
    $ 1982 "b_touch_pos≔A_Prepos_l[A_sel_v]"
    global b_touch_pos=A_Prepos_l[A_sel_v]
    $ 1983 "tilt_deg_ry≔0"
    global tilt_deg_ry=0
    $ 1984 "tilt_deg_rz≔0"
    global tilt_deg_rz=0
    $ 1985 "If b2_left_par"
    if (b2_left_par):
      $ 1986 "tilt_deg≔6"
      global tilt_deg=6
      $ 1987 "b_touch_pos≔pose_trans(b_touch_pos, p[0,0/1000,0,d2r(tilt_deg),d2r(tilt_deg_ry),d2r(tilt_deg_rz)])"
      global b_touch_pos= pose_trans (b_touch_pos, p[0,0/1000,0,d2r(tilt_deg),d2r(tilt_deg_ry),d2r(tilt_deg_rz)])
    else:
      $ 1988 "Else" "noBreak"
      $ 1989 "tilt_deg≔0.5"
      global tilt_deg=0.5
      $ 1990 "b_touch_pos≔pose_trans(b_touch_pos, p[0,0/1000,0,d2r(-tilt_deg),d2r(tilt_deg_ry),d2r(tilt_deg_rz)])"
      global b_touch_pos= pose_trans (b_touch_pos, p[0,0/1000,0,d2r(-tilt_deg),d2r(tilt_deg_ry),d2r(tilt_deg_rz)])
    end
    $ 2001 "move_pre"
    $ 2002 "If (b2_left_par≟ True  and point_dist(A_Prepos_l[A_HOR], A_Prepos_l[A_VL1])>0.032) or (b2_left_par≟ False  and point_dist(A_Prepos_l[A_HOR_R],A_Prepos_l[A_VR1])>0.032)"
    if ((b2_left_par ==   True    and  point_dist(A_Prepos_l[A_HOR], A_Prepos_l[A_VL1])>0.032)  or  (b2_left_par ==   False    and  point_dist(A_Prepos_l[A_HOR_R],A_Prepos_l[A_VR1])>0.032)):
      $ 2003 "if move from home"
      $ 2004 "j_cp≔get_actual_joint_positions()"
      global j_cp= get_actual_joint_positions ()
      $ 2005 "If b2_left_par"
      if (b2_left_par):
        $ 2006 "If norm(b_touch_pos[1]*1000)>300"
        if (norm(b_touch_pos[1]*1000)>300):
          $ 2007 "inner_p≔p[-15/1000,-35/1000,0,0,0,0]"
          global inner_p=p[-15/1000,-35/1000,0,0,0,0]
        else:
          $ 2008 "Else" "noBreak"
          $ 2009 "inner_p≔p[0,0,0,0,0,0]"
          global inner_p=p[0,0,0,0,0,0]
        end
        $ 2010 "j_tp≔get_inverse_kin(pose_add(b_touch_pos,inner_p),qnear=left_j)"
        global j_tp= get_inverse_kin (pose_add(b_touch_pos,inner_p),qnear=left_j)
      else:
        $ 2011 "Else" "noBreak"
        $ 2012 "If norm(b_touch_pos[1]*1000)>300"
        if (norm(b_touch_pos[1]*1000)>300):
          $ 2013 "inner_p≔p[-15/1000,35/1000,0,0,0,0]"
          global inner_p=p[-15/1000,35/1000,0,0,0,0]
        else:
          $ 2014 "Else" "noBreak"
          $ 2015 "inner_p≔p[0,0,0,0,0,0]"
          global inner_p=p[0,0,0,0,0,0]
        end
        $ 2016 "j_tp≔get_inverse_kin(pose_add(b_touch_pos,inner_p),qnear=right_j)"
        global j_tp= get_inverse_kin ( pose_add (b_touch_pos,inner_p),qnear=right_j)
      end
      $ 2017 "j_cp[0]=j_tp[0]"
      j_cp[0]=j_tp[0]
      $ 2018 "j_cp[1]=j_cp[1]+(j_tp[1]-j_cp[1])/2"
      j_cp[1]=j_cp[1]+(j_tp[1]-j_cp[1])/2
      $ 2019 "j_cp[2]=j_cp[2]+(j_tp[2]-j_cp[2])/2.5"
      j_cp[2]=j_cp[2]+(j_tp[2]-j_cp[2])/2.5
      $ 2020 "j_cp[3]=j_cp[3]+(j_tp[3]-j_cp[3])/2.5"
      j_cp[3]=j_cp[3]+(j_tp[3]-j_cp[3])/2.5
      $ 2021 "j_cp[4]=j_cp[4]+(j_tp[4]-j_cp[4])/3"
      j_cp[4]=j_cp[4]+(j_tp[4]-j_cp[4])/3
      $ 2022 "j_cp[5]=j_cp[5]+(j_tp[5]-j_cp[5])/1"
      j_cp[5]=j_cp[5]+(j_tp[5]-j_cp[5])/1
      $ 2023 "MoveJ"
      $ 2024 "j_cp" "breakAfter"
      movej(j_cp, a=1.3962634015954636, v=1.0471975511965976)
      $ 2025 "j_tp≔[j_cp[0],j_cp[1],j_cp[2],j_cp[3],j_tp[4],j_tp[5]]"
      global j_tp=[j_cp[0],j_cp[1],j_cp[2],j_cp[3],j_tp[4],j_tp[5]]
    end
    $ 2028 "MoveL"
    $ 2029 "b_touch_pos" "breakAfter"
    movel(pose_trans(Base, b_touch_pos), a=0.35, v=0.35)
    $ 2032 "touch_3f_down"
    $ 2034 "touch_result≔touch_fun2(b_touch_pos,b2_left_par,b9_touch_sens,b2_par_cd)"
    global touch_result=touch_fun2(b_touch_pos,b2_left_par,b9_touch_sens,b2_par_cd)
    $ 2035 "If Scallup_check≟ False "
    if (Scallup_check ==   False  ):
      $ 2036 "touch_result≔pose_trans(touch_result,p[-(Touch_dis)/1000,0,0,0,0,0])"
      global touch_result= pose_trans (touch_result,p[-(Touch_dis)/1000,0,0,0,0,0])
    else:
      $ 2037 "Else" "noBreak"
      $ 2038 "Scallup_check≔ False "
      global Scallup_check=  False
    end
    $ 2041 "A_Touch_p[A_sel_v]=touch_result"
    A_Touch_p[A_sel_v]=touch_result
    $ 2042 "If EXT_flag1[3]≟ True "
    if (EXT_flag1[3] ==   True  ):
      $ 2043 "MoveL"
      $ 2044 "manual_tp≔tilt_3f_fun(A_Touch_p[A_sel_v],basic_tilt_3f,0)"
      global manual_tp=tilt_3f_fun(A_Touch_p[A_sel_v],basic_tilt_3f,0)
      $ 2045 "manual_tp≔pose_trans(manual_tp, p[0,0,-10/1000,0,0,0])"
      global manual_tp= pose_trans (manual_tp, p[0,0,-10/1000,0,0,0])
      $ 2046 "manual_tp" "breakAfter"
      movel(pose_trans(Base, manual_tp), a=0.3, v=0.15)
      $ 2047 "Wait: 1.5"
      sleep(1.5)
    end
    $ 2048 "touch_3f_up"
    $ 2049 "If A_Prepos_l[A_sel_v_end]≟p[0,0,0,0,0,0]"
    if (A_Prepos_l[A_sel_v_end] == p[0,0,0,0,0,0]):
      $ 2050 "A_Touch_p[A_sel_v_end]=p[0,0,0,0,0,0]"
      A_Touch_p[A_sel_v_end]=p[0,0,0,0,0,0]
    else:
      $ 2051 "Else" "noBreak"
      $ 2052 "b_touch_pos≔A_Prepos_l[A_sel_v_end]"
      global b_touch_pos=A_Prepos_l[A_sel_v_end]
      $ 2053 "MoveL"
      $ 2054 "b_touch_pos" "breakAfter"
      movel(pose_trans(Base, b_touch_pos), a=0.7, v=0.5)
      $ 2055 "touch_result≔touch_fun2(b_touch_pos,b2_left_par,b9_touch_sens)"
      global touch_result=touch_fun2(b_touch_pos,b2_left_par,b9_touch_sens)
      $ 2056 "A_Touch_p[A_sel_v_end]=touch_result"
      A_Touch_p[A_sel_v_end]=touch_result
      $ 2057 "If EXT_flag1[3]≟ True "
      if (EXT_flag1[3] ==   True  ):
        $ 2058 "MoveL"
        $ 2059 "manual_tp≔A_Touch_p[A_sel_v_end]"
        global manual_tp=A_Touch_p[A_sel_v_end]
        $ 2060 "manual_tp≔tilt_3f_fun(A_Touch_p[A_sel_v_end],basic_tilt_3f,0)"
        global manual_tp=tilt_3f_fun(A_Touch_p[A_sel_v_end],basic_tilt_3f,0)
        $ 2061 "manual_tp≔pose_trans(manual_tp, p[0,0,-10/1000,0,0,0])"
        global manual_tp= pose_trans (manual_tp, p[0,0,-10/1000,0,0,0])
        $ 2062 "manual_tp" "breakAfter"
        movel(pose_trans(Base, manual_tp), a=0.3, v=0.15)
        $ 2063 "Wait: 1.5"
        sleep(1.5)
      end
    end
  end
  def weav_welding_3f():
    $ 2067 "weav_welding_3f" "noBreak"
    $ 2068 "If running_trig≟ True "
    global thread_flag_2068=0
    thread Thread_if_2068():
      $ 2069 "inv_inching(inv_inch_time)"
      inv_inching(inv_inch_time)
      $ 2070 "b_touch_pos≔A_Prepos_l[A_sel_v]"
      global b_touch_pos=A_Prepos_l[A_sel_v]
      $ 2071 "move_pre"
      $ 2072 "If (b2_left_par≟ True  and point_dist(A_Prepos_l[A_HOR], A_Prepos_l[A_VL1])>0.032) or (b2_left_par≟ False  and point_dist(A_Prepos_l[A_HOR_R],A_Prepos_l[A_VR1])>0.032)"
      if ((b2_left_par ==   True    and  point_dist(A_Prepos_l[A_HOR], A_Prepos_l[A_VL1])>0.032)  or  (b2_left_par ==   False    and  point_dist(A_Prepos_l[A_HOR_R],A_Prepos_l[A_VR1])>0.032)):
        $ 2073 "if move from home"
        $ 2074 "j_cp≔get_actual_joint_positions()"
        global j_cp= get_actual_joint_positions ()
        $ 2075 "If b2_left_par"
        if (b2_left_par):
          $ 2076 "If norm(b_touch_pos[1]*1000)>300"
          if (norm(b_touch_pos[1]*1000)>300):
            $ 2077 "inner_p≔p[-15/1000,-35/1000,0,0,0,0]"
            global inner_p=p[-15/1000,-35/1000,0,0,0,0]
          else:
            $ 2078 "Else" "noBreak"
            $ 2079 "inner_p≔p[0,0,0,0,0,0]"
            global inner_p=p[0,0,0,0,0,0]
          end
          $ 2080 "j_tp≔get_inverse_kin(pose_add(b_touch_pos,inner_p),qnear=left_j)"
          global j_tp= get_inverse_kin (pose_add(b_touch_pos,inner_p),qnear=left_j)
        else:
          $ 2081 "Else" "noBreak"
          $ 2082 "If norm(b_touch_pos[1]*1000)>300"
          if (norm(b_touch_pos[1]*1000)>300):
            $ 2083 "inner_p≔p[-15/1000,35/1000,0,0,0,0]"
            global inner_p=p[-15/1000,35/1000,0,0,0,0]
          else:
            $ 2084 "Else" "noBreak"
            $ 2085 "inner_p≔p[0,0,0,0,0,0]"
            global inner_p=p[0,0,0,0,0,0]
          end
          $ 2086 "j_tp≔get_inverse_kin(pose_add(b_touch_pos,inner_p),qnear=right_j)"
          global j_tp= get_inverse_kin ( pose_add (b_touch_pos,inner_p),qnear=right_j)
        end
        $ 2087 "j_cp[0]=j_tp[0]"
        j_cp[0]=j_tp[0]
        $ 2088 "j_cp[1]=j_cp[1]+(j_tp[1]-j_cp[1])/2"
        j_cp[1]=j_cp[1]+(j_tp[1]-j_cp[1])/2
        $ 2089 "j_cp[2]=j_cp[2]+(j_tp[2]-j_cp[2])/2.5"
        j_cp[2]=j_cp[2]+(j_tp[2]-j_cp[2])/2.5
        $ 2090 "j_cp[3]=j_cp[3]+(j_tp[3]-j_cp[3])/2.5"
        j_cp[3]=j_cp[3]+(j_tp[3]-j_cp[3])/2.5
        $ 2091 "j_cp[4]=j_cp[4]+(j_tp[4]-j_cp[4])/3"
        j_cp[4]=j_cp[4]+(j_tp[4]-j_cp[4])/3
        $ 2092 "j_cp[5]=j_cp[5]+(j_tp[5]-j_cp[5])/1"
        j_cp[5]=j_cp[5]+(j_tp[5]-j_cp[5])/1
        $ 2093 "MoveJ"
        $ 2094 "j_cp" "breakAfter"
        movej(j_cp, a=1.3962634015954636, v=1.0471975511965976)
        $ 2095 "j_tp≔[j_cp[0],j_cp[1],j_cp[2],j_cp[3],j_tp[4],j_tp[5]]"
        global j_tp=[j_cp[0],j_cp[1],j_cp[2],j_cp[3],j_tp[4],j_tp[5]]
      end
      $ 2098 "If (b2_left_par≟ True ) and (b1_cell_info_L≟A or b1_cell_info_L≟C or b1_cell_info_L≟c) and (A_sel_v≠A_VL2)"
      if ((b2_left_par ==   True  )  and  (b1_cell_info_L == A  or  b1_cell_info_L == C  or  b1_cell_info_L == c)  and  (A_sel_v != A_VL2)):
        $ 2099 "begin_3f_p≔pose_trans(A_Touch_p[A_sel_v],p[(multi_offset_z*(multi_path-1))/1000,0,0,0,0,0])"
        global begin_3f_p= pose_trans (A_Touch_p[A_sel_v],p[(multi_offset_z*(multi_path-1))/1000,0,0,0,0,0])
      else:
        $ 2100 "ElseIf (b2_left_par≟ False ) and (b1_cell_info_R≟A or b1_cell_info_R≟C or b1_cell_info_R≟c) and (A_sel_v≠A_VR2)"
        if ((b2_left_par ==   False  )  and  (b1_cell_info_R == A  or  b1_cell_info_R == C  or  b1_cell_info_R == c)  and  (A_sel_v != A_VR2)):
          $ 2101 "begin_3f_p≔pose_trans(A_Touch_p[A_sel_v],p[(multi_offset_z*(multi_path-1))/1000,0,0,0,0,0])"
          global begin_3f_p= pose_trans (A_Touch_p[A_sel_v],p[(multi_offset_z*(multi_path-1))/1000,0,0,0,0,0])
        else:
          $ 2102 "Else" "noBreak"
          $ 2103 "begin_3f_p≔A_Touch_p[A_sel_v]"
          global begin_3f_p=A_Touch_p[A_sel_v]
        end
      end
      $ 2104 "If b2_left_par≟ False "
      if (b2_left_par ==   False  ):
        $ 2105 "If (b1_cell_info_R≟c or b1_cell_info_R≟d) and A_sel_v≟A_VR2"
        if ((b1_cell_info_R == c  or  b1_cell_info_R == d)  and  A_sel_v == A_VR2):
          $ 2107 "b7_tilt_degree≔[-72,-20,15]"
          global b7_tilt_degree=[-72,-20,15]
          $ 2108 "begin_3f_p=pose_add(begin_3f_p,p[-6/1000,-1.5/1000,0,0,0,0])"
          begin_3f_p= pose_add (begin_3f_p,p[-6/1000,-1.5/1000,0,0,0,0])
          $ 2109 "a2_speed_cpm≔a2_speed_cpm*1"
          global a2_speed_cpm=a2_speed_cpm*1
          $ 2110 "a3_wv_amplitude≔a3_wv_amplitude*1"
          global a3_wv_amplitude=a3_wv_amplitude*1
          $ 2111 "a4_wv_frequency≔a4_wv_frequency*1"
          global a4_wv_frequency=a4_wv_frequency*1
          $ 2112 "b3_dealy_all≔[0,b4_wv_delay2*1,0,b6_wv_delay4*1]"
          global b3_dealy_all=[0,b4_wv_delay2*1,0,b6_wv_delay4*1]
          $ 2113 "a0_volt_ref≔a0_volt_ref*1"
          global a0_volt_ref=a0_volt_ref*1
          $ 2114 "a1_amp_ref≔a1_amp_ref*1"
          global a1_amp_ref=a1_amp_ref*1
          $ 2115 "volt and current"
          $ 2116 "squash_l≔[a0_volt_ref,a1_amp_ref,squash_enable,squash_voltage,squash_current,squash_amp,squash_speed,squash_cycle,waste_cycle,c0_offset_x,c0_offset_z]"
          global squash_l=[a0_volt_ref,a1_amp_ref,squash_enable,squash_voltage,squash_current,squash_amp,squash_speed,squash_cycle,waste_cycle,c0_offset_x,c0_offset_z]
          $ 2117 "set_current_voltage(a1_amp_ref,a0_volt_ref)"
          set_current_voltage(a1_amp_ref,a0_volt_ref)
        end
      end
      $ 2126 "welding_result = line_weaving_tp(begin_3f_p,A_Touch_p[A_sel_v_end],[a8_wv_distance,Circle_Speed,b1_appro_param,a4_wv_frequency,a3_wv_amplitude,b8_wv_type,wv_direction],b7_tilt_degree,b3_dealy_all,a9_wv_weldingon,c3_wv_arc,c7_wv_gap,a5_f_hole,b8_wv_2f,a7_weld_crater,squash_l)"
      welding_result = line_weaving_tp(begin_3f_p,A_Touch_p[A_sel_v_end],[a8_wv_distance,Circle_Speed,b1_appro_param,a4_wv_frequency,a3_wv_amplitude,b8_wv_type,wv_direction],b7_tilt_degree,b3_dealy_all,a9_wv_weldingon,c3_wv_arc,c7_wv_gap,a5_f_hole,b8_wv_2f,a7_weld_crater,squash_l)
      thread_flag_2068 = 1
    end
    if (running_trig ==   True  ):
      global thread_handler_2068=run Thread_if_2068()
      while (thread_flag_2068 == 0):
        if not(running_trig ==   True  ):
          kill thread_handler_2068
          thread_flag_2068 = 2
        else:
          sync()
        end
      end
    else:
      thread_flag_2068 = 2
    end
    $ 2127 "write_port_register(weld_done_137,1)"
    write_port_register(weld_done_137,1)
    $ 2128 "homeing()"
    homeing()
    $ 2129 "If sludge≟1"
    if (sludge == 1):
      $ 2130 "pause_trig≔ True "
      global pause_trig=  True
    end
  end
  def weav_welding_2f():
    $ 2131 "weav_welding_2f" "noBreak"
    $ 2132 "If running_trig≟ True "
    global thread_flag_2132=0
    thread Thread_if_2132():
      $ 2133 "Calculation"
      $ 2134 "If Auto_W_num[Auto_cur_cell]≟31 or Auto_W_num[Auto_cur_cell]≟32 or Auto_W_num[Auto_cur_cell]≟30"
      if (Auto_W_num[Auto_cur_cell] == 31  or  Auto_W_num[Auto_cur_cell] == 32  or  Auto_W_num[Auto_cur_cell] == 30):
        $ 2135 "cal_single"
        $ 2136 "pos_m_path≔A_Touch_p[A_HOR]"
        global pos_m_path=A_Touch_p[A_HOR]
        $ 2137 "pos_m_path_end≔A_Touch_p[A_HOR_R]"
        global pos_m_path_end=A_Touch_p[A_HOR_R]
        $ 2138 "A_middle_weld≔interpolate_pose(pos_m_path, pos_m_path_end,0.5)"
        global A_middle_weld= interpolate_pose (pos_m_path, pos_m_path_end,0.5)
      else:
        $ 2139 "Else" "noBreak"
        $ 2140 "side_offset≔10*current_path"
        global side_offset=10*current_path
        $ 2141 "side_offset≔0"
        global side_offset=0
        $ 2142 "If current_path≟2 or current_path≟4"
        if (current_path == 2  or  current_path == 4):
          $ 2143 "center_offset≔15"
          global center_offset=15
        else:
          $ 2144 "Else" "noBreak"
          $ 2145 "center_offset≔0"
          global center_offset=0
        end
        $ 2146 "cal_multi"
        $ 2147 "pos_m_path≔A_Touch_p[A_HOR]"
        global pos_m_path=A_Touch_p[A_HOR]
        $ 2148 "pos_m_path≔pose_trans(pos_m_path, p[side_offset/1000,0,0,0,0,0])"
        global pos_m_path= pose_trans (pos_m_path, p[side_offset/1000,0,0,0,0,0])
        $ 2149 "pos_m_path_end≔A_Touch_p[A_HOR_R]"
        global pos_m_path_end=A_Touch_p[A_HOR_R]
        $ 2150 "pos_m_path_end≔pose_trans(pos_m_path_end, p[-side_offset/1000,0,0,0,0,0])"
        global pos_m_path_end= pose_trans (pos_m_path_end, p[-side_offset/1000,0,0,0,0,0])
        $ 2151 "A_middle_weld≔interpolate_pose(pos_m_path, pos_m_path_end,0.5)"
        global A_middle_weld= interpolate_pose (pos_m_path, pos_m_path_end,0.5)
        $ 2152 "A_middle_weld≔pose_trans(A_middle_weld, p[-center_offset/1000,0,0,0,0,0])"
        global A_middle_weld= pose_trans (A_middle_weld, p[-center_offset/1000,0,0,0,0,0])
      end
      $ 2153 "gap_half"
      $ 2154 "gap_amp_bak≔c5_wv_gap_y"
      global gap_amp_bak=c5_wv_gap_y
      $ 2155 "gap_speed_bak≔c6_wv_gap_cpm"
      global gap_speed_bak=c6_wv_gap_cpm
      $ 2156 "gap_freq_bak≔c9_wv_gap_freq"
      global gap_freq_bak=c9_wv_gap_freq
      $ 2157 "c5_wv_gap_y≔(a3_wv_amplitude+c5_wv_gap_y)/2"
      global c5_wv_gap_y=(a3_wv_amplitude+c5_wv_gap_y)/2
      $ 2158 "c6_wv_gap_cpm≔(a2_speed_cpm+c6_wv_gap_cpm)/2"
      global c6_wv_gap_cpm=(a2_speed_cpm+c6_wv_gap_cpm)/2
      $ 2159 "c9_wv_gap_freq≔(a4_wv_frequency+c9_wv_gap_freq)/2"
      global c9_wv_gap_freq=(a4_wv_frequency+c9_wv_gap_freq)/2
      $ 2160 "c7_wv_gap≔[c4_gap_enable,c5_wv_gap_y,c6_wv_gap_cpm,c9_wv_gap_freq]"
      global c7_wv_gap=[c4_gap_enable,c5_wv_gap_y,c6_wv_gap_cpm,c9_wv_gap_freq]
      $ 2161 "Weaving"
      $ 2162 "If EXT_flag1[6]"
      if (EXT_flag1[6]):
        $ 2163 "If Auto_W_num[Auto_cur_cell]%10≟1"
        if (Auto_W_num[Auto_cur_cell]%10 == 1):
          $ 2164 "inv_inching(inv_inch_time)"
          inv_inching(inv_inch_time)
          $ 2165 "wv_direction≔1"
          global wv_direction=1
          $ 2166 "welding_result = line_weaving_tp(pos_m_path,A_middle_weld,[a8_wv_distance,Circle_Speed,b1_appro_param,a4_wv_frequency,a3_wv_amplitude,b8_wv_type,wv_direction],b7_tilt_degree,b3_dealy_all,a9_wv_weldingon,c3_wv_arc,c7_wv_gap,a5_f_hole,b8_wv_2f,a7_weld_crater,squash_l)"
          welding_result = line_weaving_tp(pos_m_path,A_middle_weld,[a8_wv_distance,Circle_Speed,b1_appro_param,a4_wv_frequency,a3_wv_amplitude,b8_wv_type,wv_direction],b7_tilt_degree,b3_dealy_all,a9_wv_weldingon,c3_wv_arc,c7_wv_gap,a5_f_hole,b8_wv_2f,a7_weld_crater,squash_l)
          $ 2167 "Wait: 0.5"
          sleep(0.5)
        end
        $ 2168 "If Auto_W_num[Auto_cur_cell]%10≟2"
        if (Auto_W_num[Auto_cur_cell]%10 == 2):
          $ 2169 "inv_inching(inv_inch_time)"
          inv_inching(inv_inch_time)
          $ 2170 "a7_weld_crater≔[d_start_current,d_start_voltage,d_start_time,d_end_current_2,d_end_voltage_2,d_end_time_2,d_lean_degree]"
          global a7_weld_crater=[d_start_current,d_start_voltage,d_start_time,d_end_current_2,d_end_voltage_2,d_end_time_2,d_lean_degree]
          $ 2171 "gap_half_right"
          $ 2172 "a3_wv_amplitude≔gap_amp_bak"
          global a3_wv_amplitude=gap_amp_bak
          $ 2173 "a2_speed_cpm≔gap_speed_bak"
          global a2_speed_cpm=gap_speed_bak
          $ 2174 "a4_wv_frequency≔gap_freq_bak"
          global a4_wv_frequency=gap_freq_bak
          $ 2175 "c7_wv_gap≔[c4_gap_enable,c5_wv_gap_y,c6_wv_gap_cpm,c9_wv_gap_freq]"
          global c7_wv_gap=[c4_gap_enable,c5_wv_gap_y,c6_wv_gap_cpm,c9_wv_gap_freq]
          $ 2176 "wv_direction≔-1"
          global wv_direction=-1
          $ 2177 "A_middle_weld≔feature_offset(A_middle_weld,p[-20/1000,0,0,0,0,0],A_Touch_p[A_sel_v])"
          global A_middle_weld=feature_offset(A_middle_weld,p[-20/1000,0,0,0,0,0],A_Touch_p[A_sel_v])
          $ 2178 "welding_result = line_weaving_tp(pos_m_path_end,A_middle_weld,[a8_wv_distance,Circle_Speed,b1_appro_param,a4_wv_frequency,a3_wv_amplitude,b8_wv_type,wv_direction],b7_tilt_degree,b3_dealy_all,a9_wv_weldingon,c3_wv_arc,c7_wv_gap,a5_f_hole,b8_wv_2f,a7_weld_crater,squash_l)"
          welding_result = line_weaving_tp(pos_m_path_end,A_middle_weld,[a8_wv_distance,Circle_Speed,b1_appro_param,a4_wv_frequency,a3_wv_amplitude,b8_wv_type,wv_direction],b7_tilt_degree,b3_dealy_all,a9_wv_weldingon,c3_wv_arc,c7_wv_gap,a5_f_hole,b8_wv_2f,a7_weld_crater,squash_l)
        end
      else:
        $ 2180 "Else" "noBreak"
        $ 2181 "If Auto_W_num[Auto_cur_cell]%10≟0"
        if (Auto_W_num[Auto_cur_cell]%10 == 0):
          $ 2182 "inv_inching(inv_inch_time)"
          inv_inching(inv_inch_time)
          $ 2183 "wv_direction≔1"
          global wv_direction=1
          $ 2184 "welding_result = line_weaving_tp(pos_m_path,pos_m_path_end,[a8_wv_distance,Circle_Speed,b1_appro_param,a4_wv_frequency,a3_wv_amplitude,b8_wv_type,wv_direction],b7_tilt_degree,b3_dealy_all,a9_wv_weldingon,c3_wv_arc,c7_wv_gap,a5_f_hole,b8_wv_2f,a7_weld_crater,squash_l)"
          welding_result = line_weaving_tp(pos_m_path,pos_m_path_end,[a8_wv_distance,Circle_Speed,b1_appro_param,a4_wv_frequency,a3_wv_amplitude,b8_wv_type,wv_direction],b7_tilt_degree,b3_dealy_all,a9_wv_weldingon,c3_wv_arc,c7_wv_gap,a5_f_hole,b8_wv_2f,a7_weld_crater,squash_l)
        else:
          $ 2185 "Else" "noBreak"
          $ 2186 "write_port_register(142,142)"
          write_port_register(142,142)
          $ 2187 "Halt"
          halt
        end
      end
      thread_flag_2132 = 1
    end
    if (running_trig ==   True  ):
      global thread_handler_2132=run Thread_if_2132()
      while (thread_flag_2132 == 0):
        if not(running_trig ==   True  ):
          kill thread_handler_2132
          thread_flag_2132 = 2
        else:
          sync()
        end
      end
    else:
      thread_flag_2132 = 2
    end
    $ 2188 "write_port_register(weld_done_137,1)"
    write_port_register(weld_done_137,1)
    $ 2189 "MoveL"
    $ 2190 "Direction: Tool Z-"
    global move_thread_flag_2190=0
    thread move_thread_2190():
      enter_critical
      move_thread_flag_2190 = 1
      local towardsPos=calculate_point_to_move_towards(get_forward_kin(), [0.0,0.0,-1.0], 0.03)
      movel(towardsPos, a=1.2, v=0.25)
      move_thread_flag_2190 = 2
      exit_critical
    end
    move_thread_flag_2190 = 0
    move_thread_han_2190 = run move_thread_2190()
    while (True):
      sleep(1.0E-10)
      if (move_thread_flag_2190 > 1):
        join move_thread_han_2190
        $ 2191 "Until (distance)"
        break
      end
      sync()
    end
    $ 2192 "homeing()"
    homeing()
    $ 2193 "If sludge≟1 or (sludge≟2 and current_path>1)"
    if (sludge == 1  or  (sludge == 2  and  current_path>1)):
      $ 2194 "If  not (Auto_W_num[Auto_cur_cell]%10≟1)"
      if (  not  (Auto_W_num[Auto_cur_cell]%10 == 1)):
        $ 2195 "pause_trig≔ True "
        global pause_trig=  True
      end
    end
  end
  def weav_welding_2f_CD():
    $ 2196 "weav_welding_2f_CD" "noBreak"
    $ 2197 "If running_trig≟ True "
    global thread_flag_2197=0
    thread Thread_if_2197():
      $ 2198 "CD_calculation"
      $ 2199 "If (Auto_W_num[Auto_cur_cell]≥100 and Auto_W_num[Auto_cur_cell]<106)  or (Auto_W_num[Auto_cur_cell]≥150 and Auto_W_num[Auto_cur_cell]<156)"
      if ((Auto_W_num[Auto_cur_cell] >= 100  and  Auto_W_num[Auto_cur_cell]<106)   or  (Auto_W_num[Auto_cur_cell] >= 150  and  Auto_W_num[Auto_cur_cell]<156)):
        $ 2200 "cal single"
        $ 2201 "cal_1"
        $ 2202 "pos_m_path_cd≔A_Touch_p[A_sel_v]"
        global pos_m_path_cd=A_Touch_p[A_sel_v]
        $ 2203 "pos_m_p_end_cd≔A_Touch_p[A_sel_v_end]"
        global pos_m_p_end_cd=A_Touch_p[A_sel_v_end]
        $ 2204 "cal_2"
        $ 2205 "pos_m_path≔A_Touch_p[A_sel_v2]"
        global pos_m_path=A_Touch_p[A_sel_v2]
        $ 2206 "pos_m_path_end≔A_Touch_p[A_sel_v_end2]"
        global pos_m_path_end=A_Touch_p[A_sel_v_end2]
        $ 2207 "A_middle_weld≔interpolate_pose(pos_m_path, pos_m_path_end,0.5)"
        global A_middle_weld= interpolate_pose (pos_m_path, pos_m_path_end,0.5)
      else:
        $ 2208 "Else" "noBreak"
        $ 2209 "cal multi"
        $ 2210 "side_offset≔0"
        global side_offset=0
        $ 2211 "If current_path≟2 or current_path≟4"
        if (current_path == 2  or  current_path == 4):
          $ 2212 "center_offset≔15"
          global center_offset=15
        else:
          $ 2213 "Else" "noBreak"
          $ 2214 "center_offset≔0"
          global center_offset=0
        end
        $ 2215 "cal_1_multi"
        $ 2216 "pos_m_path_cd≔A_Touch_p[A_sel_v]"
        global pos_m_path_cd=A_Touch_p[A_sel_v]
        $ 2217 "pos_m_path_cd≔pose_trans(pos_m_path_cd, p[side_offset/1000,0,0,0,0,0])"
        global pos_m_path_cd= pose_trans (pos_m_path_cd, p[side_offset/1000,0,0,0,0,0])
        $ 2218 "pos_m_p_end_cd≔A_Touch_p[A_sel_v_end]"
        global pos_m_p_end_cd=A_Touch_p[A_sel_v_end]
        $ 2219 "pos_m_p_end_cd≔pose_trans(pos_m_p_end_cd, p[-side_offset/1000,0,0,0,0,0])"
        global pos_m_p_end_cd= pose_trans (pos_m_p_end_cd, p[-side_offset/1000,0,0,0,0,0])
        $ 2220 "cal_2_multi"
        $ 2221 "pos_m_path≔A_Touch_p[A_sel_v2]"
        global pos_m_path=A_Touch_p[A_sel_v2]
        $ 2222 "pos_m_path≔pose_trans(pos_m_path, p[side_offset/1000,0,0,0,0,0])"
        global pos_m_path= pose_trans (pos_m_path, p[side_offset/1000,0,0,0,0,0])
        $ 2223 "pos_m_path_end≔A_Touch_p[A_sel_v_end2]"
        global pos_m_path_end=A_Touch_p[A_sel_v_end2]
        $ 2224 "pos_m_path_end≔pose_trans(pos_m_path_end, p[-side_offset/1000,0,0,0,0,0])"
        global pos_m_path_end= pose_trans (pos_m_path_end, p[-side_offset/1000,0,0,0,0,0])
        $ 2225 "A_middle_weld≔interpolate_pose(pos_m_path, pos_m_path_end,0.5)"
        global A_middle_weld= interpolate_pose (pos_m_path, pos_m_path_end,0.5)
        $ 2226 "A_middle_weld≔pose_trans(A_middle_weld, p[center_offset*wv_direction/1000,0,0,0,0,0])"
        global A_middle_weld= pose_trans (A_middle_weld, p[center_offset*wv_direction/1000,0,0,0,0,0])
      end
      $ 2227 "gap_half"
      $ 2228 "gap_amp_bak≔c5_wv_gap_y"
      global gap_amp_bak=c5_wv_gap_y
      $ 2229 "gap_speed_bak≔c6_wv_gap_cpm"
      global gap_speed_bak=c6_wv_gap_cpm
      $ 2230 "gap_freq_bak≔c9_wv_gap_freq"
      global gap_freq_bak=c9_wv_gap_freq
      $ 2231 "c5_wv_gap_y≔(a3_wv_amplitude+c5_wv_gap_y)/2"
      global c5_wv_gap_y=(a3_wv_amplitude+c5_wv_gap_y)/2
      $ 2232 "c6_wv_gap_cpm≔(a2_speed_cpm+c6_wv_gap_cpm)/2"
      global c6_wv_gap_cpm=(a2_speed_cpm+c6_wv_gap_cpm)/2
      $ 2233 "c9_wv_gap_freq≔(a4_wv_frequency+c9_wv_gap_freq)/2"
      global c9_wv_gap_freq=(a4_wv_frequency+c9_wv_gap_freq)/2
      $ 2234 "c7_wv_gap≔[c4_gap_enable,c5_wv_gap_y,c6_wv_gap_cpm,c9_wv_gap_freq]"
      global c7_wv_gap=[c4_gap_enable,c5_wv_gap_y,c6_wv_gap_cpm,c9_wv_gap_freq]
      $ 2235 "If EXT_flag1[4]≟ True  and (b1_cell_info_L≠c and b1_cell_info_L≠d and b1_cell_info_R≠c and b1_cell_info_R≠d)"
      if (EXT_flag1[4] ==   True    and  (b1_cell_info_L != c  and  b1_cell_info_L != d  and  b1_cell_info_R != c  and  b1_cell_info_R != d)):
        $ 2236 "If EXT_flag1[6]"
        if (EXT_flag1[6]):
          $ 2237 "If Auto_W_num[Auto_cur_cell]%10≟1"
          if (Auto_W_num[Auto_cur_cell]%10 == 1):
            $ 2238 "inv_inching(inv_inch_time)"
            inv_inching(inv_inch_time)
            $ 2239 "welding_result = line_weaving_tp_l(pos_m_path_cd,[pos_m_p_end_cd,pos_m_path,A_middle_weld],[a8_wv_distance,Circle_Speed,b1_appro_param,a4_wv_frequency,a3_wv_amplitude,b8_wv_type,wv_direction],b7_tilt_degree,b3_dealy_all,a9_wv_weldingon,c3_wv_arc,c7_wv_gap,a5_f_hole,b8_wv_2f,a7_weld_crater,squash_l)"
            welding_result = line_weaving_tp_l(pos_m_path_cd,[pos_m_p_end_cd,pos_m_path,A_middle_weld],[a8_wv_distance,Circle_Speed,b1_appro_param,a4_wv_frequency,a3_wv_amplitude,b8_wv_type,wv_direction],b7_tilt_degree,b3_dealy_all,a9_wv_weldingon,c3_wv_arc,c7_wv_gap,a5_f_hole,b8_wv_2f,a7_weld_crater,squash_l)
          end
          $ 2240 "If Auto_W_num[Auto_cur_cell]%10≟4"
          if (Auto_W_num[Auto_cur_cell]%10 == 4):
            $ 2241 "inv_inching(inv_inch_time)"
            inv_inching(inv_inch_time)
            $ 2242 "a7_weld_crater≔[d_start_current,d_start_voltage,d_start_time,d_end_current_2,d_end_voltage_2,d_end_time_2,d_lean_degree]"
            global a7_weld_crater=[d_start_current,d_start_voltage,d_start_time,d_end_current_2,d_end_voltage_2,d_end_time_2,d_lean_degree]
            $ 2243 "gap_half"
            $ 2244 "a3_wv_amplitude≔gap_amp_bak"
            global a3_wv_amplitude=gap_amp_bak
            $ 2245 "a2_speed_cpm≔gap_speed_bak"
            global a2_speed_cpm=gap_speed_bak
            $ 2246 "a4_wv_frequency≔gap_freq_bak"
            global a4_wv_frequency=gap_freq_bak
            $ 2247 "c7_wv_gap≔[c4_gap_enable,c5_wv_gap_y,c6_wv_gap_cpm,c9_wv_gap_freq]"
            global c7_wv_gap=[c4_gap_enable,c5_wv_gap_y,c6_wv_gap_cpm,c9_wv_gap_freq]
            $ 2248 "wv_direction≔-1*wv_direction"
            global wv_direction=-1*wv_direction
            $ 2249 "A_middle_weld≔feature_offset(A_middle_weld,p[20*wv_direction/1000,0,0,0,0,0],A_Touch_p[A_sel_v2])"
            global A_middle_weld=feature_offset(A_middle_weld,p[20*wv_direction/1000,0,0,0,0,0],A_Touch_p[A_sel_v2])
            $ 2250 "welding_result = line_weaving_tp(pos_m_path_end,A_middle_weld,[a8_wv_distance,Circle_Speed,b1_appro_param,a4_wv_frequency,a3_wv_amplitude,b8_wv_type,wv_direction],b7_tilt_degree,b3_dealy_all,a9_wv_weldingon,c3_wv_arc,c7_wv_gap,a5_f_hole,b8_wv_2f,a7_weld_crater,squash_l)"
            welding_result = line_weaving_tp(pos_m_path_end,A_middle_weld,[a8_wv_distance,Circle_Speed,b1_appro_param,a4_wv_frequency,a3_wv_amplitude,b8_wv_type,wv_direction],b7_tilt_degree,b3_dealy_all,a9_wv_weldingon,c3_wv_arc,c7_wv_gap,a5_f_hole,b8_wv_2f,a7_weld_crater,squash_l)
          end
        else:
          $ 2251 "Else" "noBreak"
          $ 2252 "If Auto_W_num[Auto_cur_cell]%10≟0"
          if (Auto_W_num[Auto_cur_cell]%10 == 0):
            $ 2253 "inv_inching(inv_inch_time)"
            inv_inching(inv_inch_time)
            $ 2254 "welding_result = line_weaving_tp_l(pos_m_path_cd,[pos_m_p_end_cd,pos_m_path,pos_m_path_end],[a8_wv_distance,Circle_Speed,b1_appro_param,a4_wv_frequency,a3_wv_amplitude,b8_wv_type,wv_direction],b7_tilt_degree,b3_dealy_all,a9_wv_weldingon,c3_wv_arc,c7_wv_gap,a5_f_hole,b8_wv_2f,a7_weld_crater,squash_l)"
            welding_result = line_weaving_tp_l(pos_m_path_cd,[pos_m_p_end_cd,pos_m_path,pos_m_path_end],[a8_wv_distance,Circle_Speed,b1_appro_param,a4_wv_frequency,a3_wv_amplitude,b8_wv_type,wv_direction],b7_tilt_degree,b3_dealy_all,a9_wv_weldingon,c3_wv_arc,c7_wv_gap,a5_f_hole,b8_wv_2f,a7_weld_crater,squash_l)
          else:
            $ 2255 "Else" "noBreak"
            $ 2256 "write_port_register(142,142)"
            write_port_register(142,142)
            $ 2257 "Halt"
            halt
          end
        end
      else:
        $ 2258 "Else" "noBreak"
        $ 2259 "If EXT_flag1[6]"
        if (EXT_flag1[6]):
          $ 2260 "If Auto_W_num[Auto_cur_cell]%10≟2"
          if (Auto_W_num[Auto_cur_cell]%10 == 2):
            $ 2261 "inv_inching(inv_inch_time)"
            inv_inching(inv_inch_time)
            $ 2262 "gap_half"
            $ 2263 "gap_amp_bak≔c5_wv_gap_y"
            global gap_amp_bak=c5_wv_gap_y
            $ 2264 "gap_speed_bak≔c6_wv_gap_cpm"
            global gap_speed_bak=c6_wv_gap_cpm
            $ 2265 "gap_freq_bak≔c9_wv_gap_freq"
            global gap_freq_bak=c9_wv_gap_freq
            $ 2266 "c5_wv_gap_y≔(a3_wv_amplitude+c5_wv_gap_y)/2"
            global c5_wv_gap_y=(a3_wv_amplitude+c5_wv_gap_y)/2
            $ 2267 "c6_wv_gap_cpm≔(a2_speed_cpm+c6_wv_gap_cpm)/2"
            global c6_wv_gap_cpm=(a2_speed_cpm+c6_wv_gap_cpm)/2
            $ 2268 "c9_wv_gap_freq≔(a4_wv_frequency+c9_wv_gap_freq)/2"
            global c9_wv_gap_freq=(a4_wv_frequency+c9_wv_gap_freq)/2
            $ 2269 "c7_wv_gap≔[c4_gap_enable,c5_wv_gap_y,c6_wv_gap_cpm,c9_wv_gap_freq]"
            global c7_wv_gap=[c4_gap_enable,c5_wv_gap_y,c6_wv_gap_cpm,c9_wv_gap_freq]
            $ 2270 "welding_result = line_weaving_tp(pos_m_path_cd,pos_m_p_end_cd,[a8_wv_distance,Circle_Speed,b1_appro_param,a4_wv_frequency,a3_wv_amplitude,b8_wv_type,wv_direction],b7_tilt_degree,b3_dealy_all,a9_wv_weldingon,c3_wv_arc,c7_wv_gap,a5_f_hole,b8_wv_2f,a7_weld_crater,squash_l)"
            welding_result = line_weaving_tp(pos_m_path_cd,pos_m_p_end_cd,[a8_wv_distance,Circle_Speed,b1_appro_param,a4_wv_frequency,a3_wv_amplitude,b8_wv_type,wv_direction],b7_tilt_degree,b3_dealy_all,a9_wv_weldingon,c3_wv_arc,c7_wv_gap,a5_f_hole,b8_wv_2f,a7_weld_crater,squash_l)
            $ 2271 "Wait: 0.5"
            sleep(0.5)
          end
          $ 2272 "If Auto_W_num[Auto_cur_cell]%10≟3"
          if (Auto_W_num[Auto_cur_cell]%10 == 3):
            $ 2273 "inv_inching(inv_inch_time)"
            inv_inching(inv_inch_time)
            $ 2274 "welding_result = line_weaving_tp(pos_m_path,A_middle_weld,[a8_wv_distance,Circle_Speed,b1_appro_param,a4_wv_frequency,a3_wv_amplitude,b8_wv_type,wv_direction],b7_tilt_degree,b3_dealy_all,a9_wv_weldingon,c3_wv_arc,c7_wv_gap,a5_f_hole,b8_wv_2f,a7_weld_crater,squash_l)"
            welding_result = line_weaving_tp(pos_m_path,A_middle_weld,[a8_wv_distance,Circle_Speed,b1_appro_param,a4_wv_frequency,a3_wv_amplitude,b8_wv_type,wv_direction],b7_tilt_degree,b3_dealy_all,a9_wv_weldingon,c3_wv_arc,c7_wv_gap,a5_f_hole,b8_wv_2f,a7_weld_crater,squash_l)
            $ 2275 "Wait: 0.5"
            sleep(0.5)
          end
          $ 2276 "If Auto_W_num[Auto_cur_cell]%10≟4"
          if (Auto_W_num[Auto_cur_cell]%10 == 4):
            $ 2277 "inv_inching(inv_inch_time)"
            inv_inching(inv_inch_time)
            $ 2278 "a7_weld_crater≔[d_start_current,d_start_voltage,d_start_time,d_end_current_2,d_end_voltage_2,d_end_time_2,d_lean_degree]"
            global a7_weld_crater=[d_start_current,d_start_voltage,d_start_time,d_end_current_2,d_end_voltage_2,d_end_time_2,d_lean_degree]
            $ 2279 "gap_half"
            $ 2280 "a3_wv_amplitude≔gap_amp_bak"
            global a3_wv_amplitude=gap_amp_bak
            $ 2281 "a2_speed_cpm≔gap_speed_bak"
            global a2_speed_cpm=gap_speed_bak
            $ 2282 "a4_wv_frequency≔gap_freq_bak"
            global a4_wv_frequency=gap_freq_bak
            $ 2283 "c7_wv_gap≔[c4_gap_enable,c5_wv_gap_y,c6_wv_gap_cpm,c9_wv_gap_freq]"
            global c7_wv_gap=[c4_gap_enable,c5_wv_gap_y,c6_wv_gap_cpm,c9_wv_gap_freq]
            $ 2284 "wv_direction≔-1*wv_direction"
            global wv_direction=-1*wv_direction
            $ 2285 "A_middle_weld≔feature_offset(A_middle_weld,p[20*wv_direction/1000,0,0,0,0,0],A_Touch_p[A_sel_v2])"
            global A_middle_weld=feature_offset(A_middle_weld,p[20*wv_direction/1000,0,0,0,0,0],A_Touch_p[A_sel_v2])
            $ 2286 "welding_result = line_weaving_tp(pos_m_path_end,A_middle_weld,[a8_wv_distance,Circle_Speed,b1_appro_param,a4_wv_frequency,a3_wv_amplitude,b8_wv_type,wv_direction],b7_tilt_degree,b3_dealy_all,a9_wv_weldingon,c3_wv_arc,c7_wv_gap,a5_f_hole,b8_wv_2f,a7_weld_crater,squash_l)"
            welding_result = line_weaving_tp(pos_m_path_end,A_middle_weld,[a8_wv_distance,Circle_Speed,b1_appro_param,a4_wv_frequency,a3_wv_amplitude,b8_wv_type,wv_direction],b7_tilt_degree,b3_dealy_all,a9_wv_weldingon,c3_wv_arc,c7_wv_gap,a5_f_hole,b8_wv_2f,a7_weld_crater,squash_l)
          end
        else:
          $ 2287 "Else" "noBreak"
          $ 2288 "If Auto_W_num[Auto_cur_cell]%10≟2"
          if (Auto_W_num[Auto_cur_cell]%10 == 2):
            $ 2289 "inv_inching(inv_inch_time)"
            inv_inching(inv_inch_time)
            $ 2290 "c7_wv_gap≔[0,c5_wv_gap_y,c6_wv_gap_cpm,c9_wv_gap_freq]"
            global c7_wv_gap=[0,c5_wv_gap_y,c6_wv_gap_cpm,c9_wv_gap_freq]
            $ 2291 "welding_result = line_weaving_tp(pos_m_path_cd,pos_m_p_end_cd,[a8_wv_distance,Circle_Speed,b1_appro_param,a4_wv_frequency,a3_wv_amplitude,b8_wv_type,wv_direction],b7_tilt_degree,b3_dealy_all,a9_wv_weldingon,c3_wv_arc,c7_wv_gap,a5_f_hole,b8_wv_2f,a7_weld_crater,squash_l)"
            welding_result = line_weaving_tp(pos_m_path_cd,pos_m_p_end_cd,[a8_wv_distance,Circle_Speed,b1_appro_param,a4_wv_frequency,a3_wv_amplitude,b8_wv_type,wv_direction],b7_tilt_degree,b3_dealy_all,a9_wv_weldingon,c3_wv_arc,c7_wv_gap,a5_f_hole,b8_wv_2f,a7_weld_crater,squash_l)
            $ 2292 "Wait: 0.5"
            sleep(0.5)
          end
          $ 2293 "If Auto_W_num[Auto_cur_cell]%10≟5"
          if (Auto_W_num[Auto_cur_cell]%10 == 5):
            $ 2294 "inv_inching(inv_inch_time)"
            inv_inching(inv_inch_time)
            $ 2295 "c7_wv_gap≔[c4_gap_enable,c5_wv_gap_y,c6_wv_gap_cpm,c9_wv_gap_freq]"
            global c7_wv_gap=[c4_gap_enable,c5_wv_gap_y,c6_wv_gap_cpm,c9_wv_gap_freq]
            $ 2296 "welding_result = line_weaving_tp(pos_m_path,pos_m_path_end,[a8_wv_distance,Circle_Speed,b1_appro_param,a4_wv_frequency,a3_wv_amplitude,b8_wv_type,wv_direction],b7_tilt_degree,b3_dealy_all,a9_wv_weldingon,c3_wv_arc,c7_wv_gap,a5_f_hole,b8_wv_2f,a7_weld_crater,squash_l)"
            welding_result = line_weaving_tp(pos_m_path,pos_m_path_end,[a8_wv_distance,Circle_Speed,b1_appro_param,a4_wv_frequency,a3_wv_amplitude,b8_wv_type,wv_direction],b7_tilt_degree,b3_dealy_all,a9_wv_weldingon,c3_wv_arc,c7_wv_gap,a5_f_hole,b8_wv_2f,a7_weld_crater,squash_l)
            $ 2297 "Wait: 0.5"
            sleep(0.5)
          end
        end
      end
      thread_flag_2197 = 1
    end
    if (running_trig ==   True  ):
      global thread_handler_2197=run Thread_if_2197()
      while (thread_flag_2197 == 0):
        if not(running_trig ==   True  ):
          kill thread_handler_2197
          thread_flag_2197 = 2
        else:
          sync()
        end
      end
    else:
      thread_flag_2197 = 2
    end
    $ 2298 "write_port_register(weld_done_137,1)"
    write_port_register(weld_done_137,1)
    $ 2302 "wv_direction≔1"
    global wv_direction=1
    $ 2303 "If Auto_W_num[Auto_cur_cell]≥150"
    if (Auto_W_num[Auto_cur_cell] >= 150):
      $ 2304 "MoveL"
      $ 2305 "Direction: Base"
      global move_thread_flag_2305=0
      thread move_thread_2305():
        enter_critical
        move_thread_flag_2305 = 1
        local towardsPos=calculate_point_to_move_towards(p[0.0,0.0,0.0,0.0,0.0,0.0], [-1,1,0.0], 0.03)
        movel(towardsPos, a=0.2, v=0.05)
        move_thread_flag_2305 = 2
        exit_critical
      end
      move_thread_flag_2305 = 0
      move_thread_han_2305 = run move_thread_2305()
      while (True):
        sleep(1.0E-10)
        if (move_thread_flag_2305 > 1):
          join move_thread_han_2305
          $ 2306 "Until (distance)"
          break
        end
        sync()
      end
    else:
      $ 2307 "ElseIf Auto_W_num[Auto_cur_cell]≥100"
      if (Auto_W_num[Auto_cur_cell] >= 100):
        $ 2308 "MoveL"
        $ 2309 "Direction: Base"
        global move_thread_flag_2309=0
        thread move_thread_2309():
          enter_critical
          move_thread_flag_2309 = 1
          local towardsPos=calculate_point_to_move_towards(p[0.0,0.0,0.0,0.0,0.0,0.0], [-1,-1,0.0], 0.03)
          movel(towardsPos, a=0.2, v=0.05)
          move_thread_flag_2309 = 2
          exit_critical
        end
        move_thread_flag_2309 = 0
        move_thread_han_2309 = run move_thread_2309()
        while (True):
          sleep(1.0E-10)
          if (move_thread_flag_2309 > 1):
            join move_thread_han_2309
            $ 2310 "Until (distance)"
            break
          end
          sync()
        end
      end
    end
    $ 2311 "MoveL"
    $ 2312 "Direction: Tool Z-"
    global move_thread_flag_2312=0
    thread move_thread_2312():
      enter_critical
      move_thread_flag_2312 = 1
      local towardsPos=calculate_point_to_move_towards(get_forward_kin(), [0.0,0.0,-1.0], 0.03)
      movel(towardsPos, a=1.2, v=0.25)
      move_thread_flag_2312 = 2
      exit_critical
    end
    move_thread_flag_2312 = 0
    move_thread_han_2312 = run move_thread_2312()
    while (True):
      sleep(1.0E-10)
      if (move_thread_flag_2312 > 1):
        join move_thread_han_2312
        $ 2313 "Until (distance)"
        break
      end
      sync()
    end
    $ 2314 "homeing()"
    homeing()
    $ 2315 "If sludge≟1 or (sludge≟2 and current_path>1)"
    if (sludge == 1  or  (sludge == 2  and  current_path>1)):
      $ 2316 "If  not (Auto_W_num[Auto_cur_cell]%10≟1 or Auto_W_num[Auto_cur_cell]%10≟2 or Auto_W_num[Auto_cur_cell]%10≟3)"
      if (  not  (Auto_W_num[Auto_cur_cell]%10 == 1  or  Auto_W_num[Auto_cur_cell]%10 == 2  or  Auto_W_num[Auto_cur_cell]%10 == 3)):
        $ 2317 "pause_trig≔ True "
        global pause_trig=  True
      end
    end
  end
  def reset_weld_param():
    $ 2318 "reset_weld_param" "noBreak"
    $ 2319 "start_num≔225"
    global start_num=225
    $ 2320 "Loop start_num<237"
    while (start_num<237):
      $ 2321 "write_port_register(start_num,0)"
      write_port_register(start_num,0)
      $ 2322 "start_num≔start_num+1"
      global start_num=start_num+1
    end
    $ 2323 "start_num≔240"
    global start_num=240
    $ 2324 "Loop start_num<256"
    while (start_num<256):
      $ 2325 "write_port_register(start_num,0)"
      write_port_register(start_num,0)
      $ 2326 "start_num≔start_num+1"
      global start_num=start_num+1
    end
  end
  def touch_sub():
    $ 2327 "touch_sub" "noBreak"
    $ 2328 "freedrive"
    $ 2329 "save_timer: Start"
    save_timer_is_counting = True
    $ 2330 "Loop save_tool≟ False  and save_timer≤0.5"
    while (get_tool_digital_in(0) ==   False    and  save_timer <= 0.5):
      $ 2331 "If save_tool≟ False "
      if (get_tool_digital_in(0) ==   False  ):
        $ 2332 "save_timer≔0"
        global save_timer=0
      end
      $ 2333 "If freedrive≟ True  and freedrive_trg≟ False "
      if (get_tool_digital_in(1) ==   True    and  freedrive_trg ==   False  ):
        $ 2334 "'Manual - Freedrive'"
        # 'Manual - Freedrive'
        $ 2335 "freedrive_mode()"
        freedrive_mode()
        $ 2336 "freedrive_trg≔ True "
        global freedrive_trg=  True
      else:
        $ 2337 "ElseIf freedrive≟ False  and freedrive_trg≟ True "
        if (get_tool_digital_in(1) ==   False    and  freedrive_trg ==   True  ):
          $ 2338 "end_freedrive_mode()"
          end_freedrive_mode()
          $ 2339 "freedrive_trg≔ False "
          global freedrive_trg=  False
        end
      end
      $ 2340 "If lamp_trig≟ False "
      if (lamp_trig ==   False  ):
        $ 2341 "lamp_trig≔ True "
        global lamp_trig=  True
      end
      $ 2342 "sync()"
      sync()
    end
    $ 2343 "save_timer: Stop"
    save_timer_is_counting = False
    $ 2344 "save_timer: Reset"
    save_timer = 0
    $ 2345 "write_port_register(touch_done_157,1)"
    write_port_register(touch_done_157,1)
    $ 2346 "Wait read_port_register(touch_done_157)≟0"
    while (not( read_port_register (touch_done_157) == 0)):
      sync()
    end
    $ 2347 "Wait save_tool=LO"
    while (get_tool_digital_in(0) == True):
      sync()
    end
  end
  $ 2 "BeforeStart"
  $ 3 "'RobotVersion'"
  # 'RobotVersion'
  $ 4 "write_port_register(160,54)"
  write_port_register(160,54)
  $ 5 "Teaching for Touch"
  $ 6 "g_current_p≔get_actual_tcp_pose()"
  global g_current_p= get_actual_tcp_pose ()
  $ 7 "MoveJ"
  $ 8 "g_current_p" "breakAfter"
  movej(g_current_p, a=1.3962634015954636, v=1.0471975511965976, r=0.05)
  $ 9 "If  False "
  if (  False  ):
    $ 10 "MoveJ"
    $ 11 "'Home'"
    # 'Home'
    $ 12 "first_p" "breakAfter"
    movej([0.6572912931442261, -1.1853707472430628, -1.1612256209002894, -2.29183799425234, 1.5053011178970337, 2.249363422393799], a=1.3962634015954636, v=1.0471975511965976)
    $ 13 "'3F Left Right'"
    # '3F Left Right'
    $ 14 "left" "breakAfter"
    movej([1.0434843552115187, -1.5100991608390455, -1.7306758129700324, -1.1948061631169296, 1.4628666284450171, 1.848321797880608], a=1.3962634015954636, v=1.0471975511965976)
    $ 15 "right" "breakAfter"
    movej([-0.10351455753530914, -1.3302576856500608, -2.115934992292752, -0.862193753976749, 1.3219395896157813, 2.4264792168573246], a=1.3962634015954636, v=1.0471975511965976)
    $ 16 "'2F Left Right'"
    # '2F Left Right'
    $ 17 "up_left" "breakAfter"
    movej([1.1752926889699076, -1.8019900427886952, -1.320977727654376, -1.5255442863405975, 1.3476341406937622, 2.041365262351603], a=1.3962634015954636, v=1.0471975511965976)
    $ 18 "up_right" "breakAfter"
    movej([-0.490858516659304, -1.5854285429454542, -1.6450882962874376, -1.2830655228732084, 1.6157391701919699, 1.9100727821897805], a=1.3962634015954636, v=1.0471975511965976)
    $ 19 "Packing_pos" "breakAfter"
    movej([1.5877798795700073, -0.0173419157611292, -2.4983108679400843, -1.4065726439105433, 1.626846194267273, 3.0169763565063477], a=1.3962634015954636, v=1.0471975511965976)
    $ 20 "pre_position" "breakAfter"
    movej([1.2637099027633667, -0.695505444203512, -2.0481718222247522, -1.9413569609271448, 2.573765277862549, 1.3775802850723267], a=1.3962634015954636, v=1.0471975511965976)
    $ 21 "middle_pos" "breakAfter"
    movej([-1.8762093791333925, -1.0408674059020342, -1.3551139327963426, -1.843592441478755, 1.9056326083560464, 0.7075109167810423], a=1.3962634015954636, v=1.0471975511965976)
    $ 22 "Mounting_pos" "breakAfter"
    movej([0.6231353085164267, -0.6300961531972575, -0.9034285948871803, -1.770059340221131, 1.417516049558281, 1.7792033261567348], a=1.3962634015954636, v=1.0471975511965976)
    $ 23 "pre_mounting" "breakAfter"
    movej([1.2356762886047363, -0.8703244368182581, -0.942230526600973, -2.3905327955829065, 1.3216267824172974, 2.6514604091644287], a=1.3962634015954636, v=1.0471975511965976)
    $ 24 "'firstly touch center and side, side_L is side touch pose'"
    # 'firstly touch center and side, side_L is side touch pose'
    $ 25 "side_p_L" "breakAfter"
    movej([0.7063748268745771, -1.3604975314992132, -1.990433834727808, -1.0668367667667118, 1.6921872781537495, 1.2509236145111355], a=1.3962634015954636, v=1.0471975511965976)
    $ 26 "side_p_R" "breakAfter"
    movej([0.05431400611996651, -1.4896310011493128, -1.8839471975909632, -1.079590145741598, 1.21127450466156, 2.729013204574585], a=1.3962634015954636, v=1.0471975511965976)
    $ 27 "left_prep_p" "breakAfter"
    movej([0.7465318441390991, -0.9293935934649866, -1.54653245607485, -2.120742146168844, 1.6612900495529175, 1.4639835357666016], a=1.3962634015954636, v=1.0471975511965976)
    $ 28 "right_prep_p" "breakAfter"
    movej([0.07502574473619461, -0.9044721762286585, -1.5771153608905237, -1.9135711828814905, 1.726387619972229, 2.67875337600708], a=1.3962634015954636, v=1.0471975511965976)
    $ 29 "top_right" "breakAfter"
    movej([-0.02242371234582219, -0.9682979219978707, -1.1486403794481532, -1.814672356578109, 1.0564512116488283, 1.9516847799391646], a=1.3962634015954636, v=1.0471975511965976)
    $ 30 "down_right" "breakAfter"
    movej([-0.10387097169690396, -0.8634965401570085, -1.6224404602167288, -1.9527388322769834, 1.2604034373302166, 1.9362943911099855], a=1.3962634015954636, v=1.0471975511965976)
    $ 31 "way_600_3F_VL1" "breakAfter"
    movej([1.4495428629911409, -0.8691188832486789, -1.6280015865128723, -1.109862842185814, 0.958613460846621, 1.8600136596738885], a=1.3962634015954636, v=1.0471975511965976)
    $ 32 "way_3F_42" "breakAfter"
    movej([0.36805654405146704, -0.7862968504575107, -2.173257016154224, -1.4479178800416523, 0.8821879504915225, 2.8855763836420314], a=1.3962634015954636, v=1.0471975511965976)
    $ 33 "Waypoint_3" "breakAfter"
    movej([1.1380372507706311, -0.9407851141189099, -1.233329099346161, -2.2390373632318763, 1.2601061328687342, 1.8320151492624872], a=1.3962634015954636, v=1.0471975511965976)
  end
  $ 34 "waypoint"
  $ 35 "first_p_wp≔first_p"
  global first_p_wp=p[.431245807847, -.007259877891, .087796870964, 2.814824648791, -.024151220978, 1.380109909682]
  $ 36 "home_pos_j≔get_inverse_kin(first_p,qnear=[0.788235068321228, -1.101443115864889, -1.2219904104815882, -2.3243168036090296, 1.506469488143921, 2.3651483058929443])"
  global home_pos_j= get_inverse_kin (p[.431245807847, -.007259877891, .087796870964, 2.814824648791, -.024151220978, 1.380109909682],qnear=[0.788235068321228, -1.101443115864889, -1.2219904104815882, -2.3243168036090296, 1.506469488143921, 2.3651483058929443])
  $ 37 "left_j≔get_inverse_kin(left,qnear=[1.0260889556530308, -1.5106289215345097, -1.741216762689402, -1.178962336228949, 1.4987324920877318, 1.8103628938054515])"
  global left_j= get_inverse_kin (p[.480496318984, .411279115151, .006998291210, -2.211681476386, -.899147924387, -1.383032568605],qnear=[1.0260889556530308, -1.5106289215345097, -1.741216762689402, -1.178962336228949, 1.4987324920877318, 1.8103628938054515])
  $ 38 "right_j≔get_inverse_kin(right,qnear=[-0.04005625546610858, -1.5553040811514833, -1.9086689348599588, -0.877043115030812, 1.298887151057777, 2.511237649551841])"
  global right_j= get_inverse_kin (p[.475000000000, -.421403215678, .026417194146, 1.917761036827, -1.141682393512, 1.523356199292],qnear=[-0.04005625546610858, -1.5553040811514833, -1.9086689348599588, -0.877043115030812, 1.298887151057777, 2.511237649551841])
  $ 39 "left_prep_p_v≔left_prep_p"
  global left_prep_p_v=p[.305384281395, .209992212444, .052849493181, -2.261254200610, -.979668861910, -1.115042887278]
  $ 40 "right_prep_p_v≔right_prep_p"
  global right_prep_p_v=p[.351918991358, -.200990531927, .062804013870, 2.289356494782, -1.513598216236, 1.281039242610]
  $ 41 "Packing_pos_wp≔Packing_pos"
  global Packing_pos_wp=p[.278714911898, .357008020042, .025408199530, -2.146966801259, .195978635494, -.919933898512]
  $ 42 "pre_position_wp≔pre_position"
  global pre_position_wp=p[-.206981089246, .377817475970, .184983176991, -1.570600793609, -.863923490888, -.089005332274]
  $ 43 "pre_mounting_wp≔pre_mounting"
  global pre_mounting_wp=p[.460443249232, .114922015113, .277198878359, -2.240057458299, .067416497001, -1.614091004704]
  $ 44 "mounting_wp≔Mounting_pos"
  global mounting_wp=p[.365658114054, -.003207132620, .718667154922, -1.220752075696, -.066673751622, -2.363385143972]
  $ 45 "Setting"
  $ 46 "inv_inch_time≔0.4"
  global inv_inch_time=0.4
  $ 47 "a7_cell_bottom≔-50.2"
  global a7_cell_bottom=-50.2
  $ 48 "get_center≔470"
  global get_center=470
  $ 49 "work_touch_dis≔50"
  global work_touch_dis=50
  $ 50 "cd_extra_dis≔6"
  global cd_extra_dis=6
  $ 51 "side_pos_x≔-10"
  global side_pos_x=-10
  $ 52 "sec_touch_dis≔35"
  global sec_touch_dis=35
  $ 53 "Touch_dis≔30"
  global Touch_dis=30
  $ 54 "offset_2f_begin≔5"
  global offset_2f_begin=5
  $ 55 "offset_3f_begin≔5"
  global offset_3f_begin=5
  $ 56 "multi_offset_z≔3"
  global multi_offset_z=3
  $ 57 "simulation_mode≔ False "
  global simulation_mode=  False
  $ 58 "tilt_deg_man≔7"
  global tilt_deg_man=7
  $ 59 "Initialization"
  $ 60 "reset_revolution_counter()"
  reset_revolution_counter()
  $ 61 "get_center_bak≔get_center"
  global get_center_bak=get_center
  $ 62 "welding_program≔ False "
  global welding_program=  False
  $ 63 "vr2_p1≔p[0,0,0,0,0,0]"
  global vr2_p1=p[0,0,0,0,0,0]
  $ 64 "running_trig≔ False "
  global running_trig=  False
  $ 65 "pb_comm_count≔0"
  global pb_comm_count=0
  $ 66 "pendant_hb≔read_port_register(161)"
  global pendant_hb= read_port_register (161)
  $ 67 "pause_trig≔ False "
  global pause_trig=  False
  $ 68 "multi_path≔1"
  global multi_path=1
  $ 69 "reset_trig≔ False "
  global reset_trig=  False
  $ 70 "heartbeat≔0"
  global heartbeat=0
  $ 71 "back_2f≔ False "
  global back_2f=  False
  $ 72 "t_time≔0"
  global t_time=0
  $ 73 "cd_offset≔35"
  global cd_offset=35
  $ 74 "write_port_register(144,0)"
  write_port_register(144,0)
  $ 75 "time_cal_trig≔ False "
  global time_cal_trig=  False
  $ 76 "current_2f≔0"
  global current_2f=0
  $ 77 "A_cur_2f≔0"
  global A_cur_2f=0
  $ 78 "CD_MLR≔ True "
  global CD_MLR=  True
  $ 79 "auto_on≔ False "
  global auto_on=  False
  $ 80 "event_cal_on≔ False "
  global event_cal_on=  False
  $ 81 "event_side_on≔ False "
  global event_side_on=  False
  $ 82 "Auto_trig≔ False "
  global Auto_trig=  False
  $ 83 "lamp_trig≔ False "
  global lamp_trig=  False
  $ 84 "calcu_trig≔ False "
  global calcu_trig=  False
  $ 85 "current_path≔1"
  global current_path=1
  $ 86 "freedrive_trg≔ False "
  global freedrive_trg=  False
  $ 87 "Inch_trg≔ False "
  global Inch_trg=  False
  $ 88 "wv_direction≔1"
  global wv_direction=1
  $ 89 "Move_trig≔ False "
  global Move_trig=  False
  $ 90 "CELL_ROBOT_DIST≔500"
  global CELL_ROBOT_DIST=500
  $ 91 "CELL_WIDTH≔700"
  global CELL_WIDTH=700
  $ 92 "CELL_BOTTOM≔a7_cell_bottom"
  global CELL_BOTTOM=a7_cell_bottom
  $ 93 "scallop_info≔ False "
  global scallop_info=  False
  $ 94 "Carl_info≔ False "
  global Carl_info=  False
  $ 95 "touch_done_2f≔ False "
  global touch_done_2f=  False
  $ 96 "get_pose_side≔0"
  global get_pose_side=0
  $ 97 "get_pose_side_t≔0"
  global get_pose_side_t=0
  $ 98 "ba_trig≔ False "
  global ba_trig=  False
  $ 99 "touch_m_check≔0"
  global touch_m_check=0
  $ 100 "basic_tilt_2f≔[30,5,0]"
  global basic_tilt_2f=[30,5,0]
  $ 102 "basic_tilt_3f≔[0,-27,0]"
  global basic_tilt_3f=[0,-27,0]
  $ 104 "modbus_name"
  $ 105 "weld_done_137≔137"
  global weld_done_137=137
  $ 106 "robot_ready_141≔141"
  global robot_ready_141=141
  $ 107 "cell_3f_2f_151≔151"
  global cell_3f_2f_151=151
  $ 108 "cell_info_152≔152"
  global cell_info_152=152
  $ 109 "weld_req_153≔153"
  global weld_req_153=153
  $ 110 "touch_cell_155≔155"
  global touch_cell_155=155
  $ 111 "touch_num_156≔156"
  global touch_num_156=156
  $ 112 "touch_done_157≔157"
  global touch_done_157=157
  $ 113 "robot_move_163≔163"
  global robot_move_163=163
  $ 114 "robot_pose_164≔164"
  global robot_pose_164=164
  $ 115 "work_type_165≔165"
  global work_type_165=165
  $ 116 "arc_onoff_168≔168"
  global arc_onoff_168=168
  $ 117 "beforeafter_170≔170"
  global beforeafter_170=170
  $ 118 "return_done_240≔240"
  global return_done_240=240
  $ 119 "a0_Job_Mode≔0"
  global a0_Job_Mode=0
  $ 120 "position_3F≔1"
  global position_3F=1
  $ 121 "position_2F≔2"
  global position_2F=2
  $ 122 "cell_par"
  $ 123 "A≔1"
  global A=1
  $ 124 "B≔2"
  global B=2
  $ 125 "C≔3"
  global C=3
  $ 126 "c≔4"
  global c=4
  $ 127 "D≔5"
  global D=5
  $ 128 "d≔6"
  global d=6
  $ 129 "E≔7"
  global E=7
  $ 130 "e≔8"
  global e=8
  $ 131 "A_VL1≔1"
  global A_VL1=1
  $ 132 "A_VL2≔2"
  global A_VL2=2
  $ 133 "A_VR1≔3"
  global A_VR1=3
  $ 134 "A_VR2≔4"
  global A_VR2=4
  $ 135 "A_HOR≔5"
  global A_HOR=5
  $ 136 "A_HOR_R≔7"
  global A_HOR_R=7
  $ 137 "A_HOR_ML≔6"
  global A_HOR_ML=6
  $ 138 "A_HOR_MR≔8"
  global A_HOR_MR=8
  $ 139 "A_HOR_M≔9"
  global A_HOR_M=9
  $ 140 "A_VL1_END≔10"
  global A_VL1_END=10
  $ 141 "A_VL2_END≔11"
  global A_VL2_END=11
  $ 142 "A_VR1_END≔12"
  global A_VR1_END=12
  $ 143 "A_VR2_END≔13"
  global A_VR2_END=13
  $ 144 "A_HOR_2path≔14"
  global A_HOR_2path=14
  $ 145 "A_HOR_3path≔15"
  global A_HOR_3path=15
  $ 146 "A_HOR_4path≔16"
  global A_HOR_4path=16
  $ 147 "A_HOR_2path_CD≔17"
  global A_HOR_2path_CD=17
  $ 148 "A_HOR_3path_CD≔18"
  global A_HOR_3path_CD=18
  $ 149 "A_HOR_4path_CD≔19"
  global A_HOR_4path_CD=19
  $ 150 "Script: UR_samho_weaving_V7.0_CB.script"
  wv_wp1 = p[0,0,0,0,0,0]
  dumy_p = p[0,0,0,0,0,0]
  global background_cal = 0
  global background_pose = [dumy_p,dumy_p,dumy_p,dumy_p]
  global background_ready = 0
  global timer_counter = 0
  global timer_counting = False
  global wcr_counter = 0
  global wcr_counting = False
  global get_wcr = False
  global arc_sens_onoff = 0
  global welding_off_t = 55
  global weld_onoff = False
  global isHicomm = True
  global isTouchWCR = True
  global welding_program = False
  global arc_sens_2F = False

  thread thread_timer():
    error_time = 5
    start_gas_time = 2
    while (True):
      if (timer_counting):
        timer_counter = timer_counter + get_steptime()
        write_output_float_register(0,timer_counter)

        get_wcr = read_welder(5)
        weld_onoff = read_welder_control(0)

        welding_off_t = read_port_register(168)
        if(get_wcr):
          global arc_sens_onoff = 1
        else:
          global arc_sens_onoff = 0
        end
        if(get_wcr and welding_off_t == 2 and weld_onoff == True):
          wcr_counter=0
        elif(wcr_counter>(error_time+start_gas_time) and welding_off_t == 2 and weld_onoff == True):
          write_port_register(202,0)
          write_port_register(149,0)
          write_welder(0,False)
          set_standard_digital_out(0,False)
          write_port_register(142,131)
          sleep(0.5)
          halt
        elif(get_wcr == False and welding_off_t == 2 and weld_onoff == True):
          wcr_counter = wcr_counter + get_steptime()
        end
      end
      sync()
    end
  end

  def RTDE_init():
    # timer
    write_output_float_register(0,0)
    # WCR IN
    write_output_float_register(1,0)
    # Welding Current
    write_output_float_register(2,0)
    # Welding Voltage
    write_output_float_register(3,0)
    # X offset
    write_output_float_register(4,0)
    # Z offset
    write_output_float_register(5,0)
    # PLUS Integral
    write_output_float_register(6,0)
    # MINUS Integral
    write_output_float_register(7,0)
    # Standard_Arc_Current
    write_output_float_register(8,0)
    # ALL Integral
    write_output_float_register(9,0)
    # x up
    write_output_float_register(10,0)
    # x ui
    write_output_float_register(11,0)
    # z up
    write_output_float_register(12,0)
    # z ui
    write_output_float_register(13,0)
    # x
    write_output_float_register(14,0)
    # y
    write_output_float_register(15,0)
    # z
    write_output_float_register(16,0)
    # welding on/off polyscope
    write_output_float_register(17,0)
    # touch on/off polyscope
    write_output_float_register(18,0)
    # ratio_t
    write_output_float_register(19,0)
    # get_wcr polyscope
    write_output_float_register(20,0)
    # get_touch polyscope
    write_output_float_register(21,0)
    # write_welder
    write_output_float_register(22,0)
    # MIDDLE_Integral_org
    write_output_float_register(23,0)
    # PLUS Integral_org
    write_output_float_register(24,0)
    # MINUS Integral_org
    write_output_float_register(25,0)

    #init
    global cycle_number = 0
    global cycle_done = False
    global cycle1_plus = 0
    global cycle1_minus = 0
    global cycle1_middle = 0
    global current_to_welding_m = read_port_register(133)
    global voltage_to_welding_m = read_port_register(134)/10
    global c_maxcut = current_to_welding_m*1.2
    global c_mincut = current_to_welding_m*0.8
    global v_maxcut = voltage_to_welding_m*1.2
    global v_mincut = voltage_to_welding_m*0.8
    global Standard_Arc_Current = current_to_welding_m
    global Standard_Arc_voltage = voltage_to_welding_m
    global FB_CURRENT_UR = 0
    global FB_VOLTAGE_UR = 0
    global FB_CURRENT_UR_org = 0
    global FB_VOLTAGE_UR_org = 0
    global one_cycle_p_count = 0
    global one_cycle_m_count = 0
    global one_cycle_p_accum = 0
    global one_cycle_m_accum = 0
    global one_cycle_p_accum_org = 0
    global one_cycle_m_accum_org = 0
    global cal_off_ang_rx = 0
    global cal_off_ang_ry = 0
    global Up = 0
    global Ui = 0
    global Pi_sum = 0
    global Up_z = 0
    global Ui_z = 0
    global Pi_sum_z = 0
    global peak_value = 0
    global ratio_t = 0
    global welding_off_t = 55
    global program_weld_on = False
    global next_path_c = False
    global move_p = [dumy_p,dumy_p,dumy_p,dumy_p]
    global hicomm = True
    global current_on = False
    timer_counter = 0
    sync()
  end

  # get line distance without caring orientation
  def get_line_dist(get_wp1,get_wp2):
    return sqrt((get_wp2[0]-get_wp1[0])*(get_wp2[0]-get_wp1[0])+(get_wp2[1]-get_wp1[1])*(get_wp2[1]-get_wp1[1])+(get_wp2[2]-get_wp1[2])*(get_wp2[2]-get_wp1[2]))
  end

  def plus_minus(num):
    if(num<0):
      return -1
    else:
      return 1
    end
  end

  def get_feature_plane_xz(p1, p2, p3):

    # Step 1. Get the direction vectors
    d12 = [ p2[0]-p1[0], p2[1]-p1[1], p2[2]-p1[2] ]
    d13 = [ p3[0]-p1[0], p3[1]-p1[1], p3[2]-p1[2] ]

    # Step 2. Get the direction vector of Z axis by cross product of d12 and d13
    dy = cross_product(d13, d12)

    # Step 3. Get the X and Z unit direction vectors by normalizing d12 and dz
    temp = norm(d12)
    ux = [ d12[0]/temp, d12[1]/temp, d12[2]/temp ]
    temp = norm(dy)
    uy = [ dy[0]/temp, dy[1]/temp, dy[2]/temp ]

    # Step 4. Get Y unit direction vector by cross product of uz and ux
    uz = cross_product(ux, uy)

    # Step 5. Get the rotation matrix from the unit direction vectors
    rotmat = [ ux[0], ux[1], ux[2], uy[0], uy[1], uy[2], uz[0], uz[1], uz[2] ]

    # Step 6. Get the rotation vector from the rotation matrix
    rotvec = rotmat2rotvec(rotmat)

